Fanuc TP program (LS listing): layer_8.ls

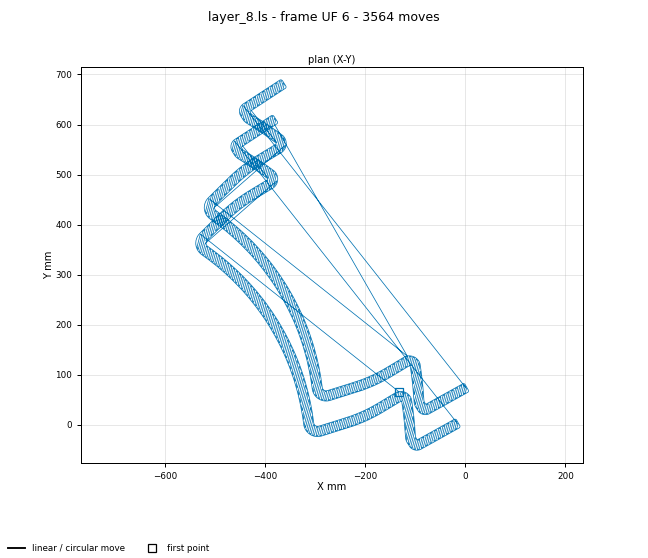
[picture p0: tool path of layer_8.ls in frame UF 6, 3564 of 3564 moves have a stored position in this frame; points joined in program order, loops and branches not executed]
/PROG layer_8
/ATTR
OWNER       = MNEDITOR;
CREATE      = DATE 100-11-20  TIME 09:43:21;
MODIFIED    = DATE 100-12-05  TIME 05:26:29;
LINE_COUNT = 1792;
PROTECT     = READ_WRITE;
TCD:  STACK_SIZE    = 0,
      TASK_PRIORITY = 50,
      TIME_SLICE    = 0,
      BUSY_LAMP_OFF = 0,
      ABORT_REQUEST = 0,
      PAUSE_REQUEST = 0;
DEFAULT_GROUP   = 1,1,*,*,*;
CONTROL_CODE    = 00000000 00000000;
/MN
:R[35]=79.0;
:R[34]=0;
1: L P[1] 240cm/min CNT100 COORD ;
: Arc Start[1];
2: L P[2] 240cm/min CNT100 COORD PTH ;
3: L P[3] 240cm/min CNT100 COORD PTH ;
4: L P[4] 240cm/min CNT100 COORD PTH ;
5: L P[5] 240cm/min CNT100 COORD PTH ;
6: L P[6] 240cm/min CNT100 COORD PTH ;
7: L P[7] 240cm/min CNT100 COORD PTH ;
8: L P[8] 240cm/min CNT100 COORD PTH ;
9: L P[9] 240cm/min CNT100 COORD PTH ;
10: L P[10] 240cm/min CNT100 COORD PTH ;
11: L P[11] 240cm/min CNT100 COORD PTH ;
12: L P[12] 240cm/min CNT100 COORD PTH ;
13: L P[13] 240cm/min CNT100 COORD PTH ;
14: L P[14] 240cm/min CNT100 COORD PTH ;
15: L P[15] 240cm/min CNT100 COORD PTH ;
16: L P[16] 240cm/min CNT100 COORD PTH ;
17: L P[17] 240cm/min CNT100 COORD PTH ;
18: L P[18] 240cm/min CNT100 COORD PTH ;
19: L P[19] 240cm/min CNT100 COORD PTH ;
20: L P[20] 240cm/min CNT100 COORD PTH ;
21: L P[21] 240cm/min CNT100 COORD PTH ;
22: L P[22] 240cm/min CNT100 COORD PTH ;
23: L P[23] 240cm/min CNT100 COORD PTH ;
24: L P[24] 240cm/min CNT100 COORD PTH ;
25: L P[25] 240cm/min CNT100 COORD PTH ;
26: L P[26] 240cm/min CNT100 COORD PTH ;
27: L P[27] 240cm/min CNT100 COORD PTH ;
28: L P[28] 240cm/min CNT100 COORD PTH ;
29: L P[29] 240cm/min CNT100 COORD PTH ;
30: L P[30] 240cm/min CNT100 COORD PTH ;
31: L P[31] 240cm/min CNT100 COORD PTH ;
32: L P[32] 240cm/min CNT100 COORD PTH ;
33: L P[33] 240cm/min CNT100 COORD PTH ;
34: L P[34] 240cm/min CNT100 COORD PTH ;
35: L P[35] 240cm/min CNT100 COORD PTH ;
36: L P[36] 240cm/min CNT100 COORD PTH ;
37: L P[37] 240cm/min CNT100 COORD PTH ;
38: L P[38] 240cm/min CNT100 COORD PTH ;
39: L P[39] 240cm/min CNT100 COORD PTH ;
40: L P[40] 240cm/min CNT100 COORD PTH ;
41: L P[41] 240cm/min CNT100 COORD PTH ;
42: L P[42] 240cm/min CNT100 COORD PTH ;
43: L P[43] 240cm/min CNT100 COORD PTH ;
44: L P[44] 240cm/min CNT100 COORD PTH ;
45: L P[45] 240cm/min CNT100 COORD PTH ;
46: L P[46] 240cm/min CNT100 COORD PTH ;
47: L P[47] 240cm/min CNT100 COORD PTH ;
48: L P[48] 240cm/min CNT100 COORD PTH ;
49: L P[49] 240cm/min CNT100 COORD PTH ;
50: L P[50] 240cm/min CNT100 COORD PTH ;
51: L P[51] 240cm/min CNT100 COORD PTH ;
52: L P[52] 240cm/min CNT100 COORD PTH ;
53: L P[53] 240cm/min CNT100 COORD PTH ;
54: L P[54] 240cm/min CNT100 COORD PTH ;
55: L P[55] 240cm/min CNT100 COORD PTH ;
56: L P[56] 240cm/min CNT100 COORD PTH ;
57: L P[57] 240cm/min CNT100 COORD PTH ;
58: L P[58] 240cm/min CNT100 COORD PTH ;
59: L P[59] 240cm/min CNT100 COORD PTH ;
60: L P[60] 240cm/min CNT100 COORD PTH ;
61: L P[61] 240cm/min CNT100 COORD PTH ;
62: L P[62] 240cm/min CNT100 COORD PTH ;
63: L P[63] 240cm/min CNT100 COORD PTH ;
64: L P[64] 240cm/min CNT100 COORD PTH ;
65: L P[65] 240cm/min CNT100 COORD PTH ;
66: L P[66] 240cm/min CNT100 COORD PTH ;
67: L P[67] 240cm/min CNT100 COORD PTH ;
68: L P[68] 240cm/min CNT100 COORD PTH ;
69: L P[69] 240cm/min CNT100 COORD PTH ;
70: L P[70] 240cm/min CNT100 COORD PTH ;
71: L P[71] 240cm/min CNT100 COORD PTH ;
72: L P[72] 240cm/min CNT100 COORD PTH ;
73: L P[73] 240cm/min CNT100 COORD PTH ;
74: L P[74] 240cm/min CNT100 COORD PTH ;
75: L P[75] 240cm/min CNT100 COORD PTH ;
76: L P[76] 240cm/min CNT100 COORD PTH ;
77: L P[77] 240cm/min CNT100 COORD PTH ;
78: L P[78] 240cm/min CNT100 COORD PTH ;
79: L P[79] 240cm/min CNT100 COORD PTH ;
80: L P[80] 240cm/min CNT100 COORD PTH ;
81: L P[81] 240cm/min CNT100 COORD PTH ;
82: L P[82] 240cm/min CNT100 COORD PTH ;
83: L P[83] 240cm/min CNT100 COORD PTH ;
84: L P[84] 240cm/min CNT100 COORD PTH ;
85: L P[85] 240cm/min CNT100 COORD PTH ;
86: L P[86] 240cm/min CNT100 COORD PTH ;
87: L P[87] 240cm/min CNT100 COORD PTH ;
88: L P[88] 240cm/min CNT100 COORD PTH ;
89: L P[89] 240cm/min CNT100 COORD PTH ;
90: L P[90] 240cm/min CNT100 COORD PTH ;
91: L P[91] 240cm/min CNT100 COORD PTH ;
92: L P[92] 240cm/min CNT100 COORD PTH ;
93: L P[93] 240cm/min CNT100 COORD PTH ;
94: L P[94] 240cm/min CNT100 COORD PTH ;
95: L P[95] 240cm/min CNT100 COORD PTH ;
96: L P[96] 240cm/min CNT100 COORD PTH ;
97: L P[97] 240cm/min CNT100 COORD PTH ;
98: L P[98] 240cm/min CNT100 COORD PTH ;
99: L P[99] 240cm/min CNT100 COORD PTH ;
100: L P[100] 240cm/min CNT100 COORD PTH ;
101: L P[101] 240cm/min CNT100 COORD PTH ;
102: L P[102] 240cm/min CNT100 COORD PTH ;
103: L P[103] 240cm/min CNT100 COORD PTH ;
104: L P[104] 240cm/min CNT100 COORD PTH ;
105: L P[105] 240cm/min CNT100 COORD PTH ;
106: L P[106] 240cm/min CNT100 COORD PTH ;
107: L P[107] 240cm/min CNT100 COORD PTH ;
108: L P[108] 240cm/min CNT100 COORD PTH ;
109: L P[109] 240cm/min CNT100 COORD PTH ;
110: L P[110] 240cm/min CNT100 COORD PTH ;
111: L P[111] 240cm/min CNT100 COORD PTH ;
112: L P[112] 240cm/min CNT100 COORD PTH ;
113: L P[113] 240cm/min CNT100 COORD PTH ;
114: L P[114] 240cm/min CNT100 COORD PTH ;
115: L P[115] 240cm/min CNT100 COORD PTH ;
116: L P[116] 240cm/min CNT100 COORD PTH ;
117: L P[117] 240cm/min CNT100 COORD PTH ;
118: L P[118] 240cm/min CNT100 COORD PTH ;
119: L P[119] 240cm/min CNT100 COORD PTH ;
120: L P[120] 240cm/min CNT100 COORD PTH ;
121: L P[121] 240cm/min CNT100 COORD PTH ;
122: L P[122] 240cm/min CNT100 COORD PTH ;
123: L P[123] 240cm/min CNT100 COORD PTH ;
124: L P[124] 240cm/min CNT100 COORD PTH ;
125: L P[125] 240cm/min CNT100 COORD PTH ;
126: L P[126] 240cm/min CNT100 COORD PTH ;
127: L P[127] 240cm/min CNT100 COORD PTH ;
128: L P[128] 240cm/min CNT100 COORD PTH ;
129: L P[129] 240cm/min CNT100 COORD PTH ;
130: L P[130] 240cm/min CNT100 COORD PTH ;
131: L P[131] 240cm/min CNT100 COORD PTH ;
132: L P[132] 240cm/min CNT100 COORD PTH ;
133: L P[133] 240cm/min CNT100 COORD PTH ;
134: L P[134] 240cm/min CNT100 COORD PTH ;
135: L P[135] 240cm/min CNT100 COORD PTH ;
136: L P[136] 240cm/min CNT100 COORD PTH ;
137: L P[137] 240cm/min CNT100 COORD PTH ;
138: L P[138] 240cm/min CNT100 COORD PTH ;
139: L P[139] 240cm/min CNT100 COORD PTH ;
140: L P[140] 240cm/min CNT100 COORD PTH ;
141: L P[141] 240cm/min CNT100 COORD PTH ;
142: L P[142] 240cm/min CNT100 COORD PTH ;
143: L P[143] 240cm/min CNT100 COORD PTH ;
144: L P[144] 240cm/min CNT100 COORD PTH ;
145: L P[145] 240cm/min CNT100 COORD PTH ;
146: L P[146] 240cm/min CNT100 COORD PTH ;
147: L P[147] 240cm/min CNT100 COORD PTH ;
148: L P[148] 240cm/min CNT100 COORD PTH ;
149: L P[149] 240cm/min CNT100 COORD PTH ;
150: L P[150] 240cm/min CNT100 COORD PTH ;
151: L P[151] 240cm/min CNT100 COORD PTH ;
152: L P[152] 240cm/min CNT100 COORD PTH ;
153: L P[153] 240cm/min CNT100 COORD PTH ;
154: L P[154] 240cm/min CNT100 COORD PTH ;
155: L P[155] 240cm/min CNT100 COORD PTH ;
156: L P[156] 240cm/min CNT100 COORD PTH ;
157: L P[157] 240cm/min CNT100 COORD PTH ;
158: L P[158] 240cm/min CNT100 COORD PTH ;
159: L P[159] 240cm/min CNT100 COORD PTH ;
160: L P[160] 240cm/min CNT100 COORD PTH ;
161: L P[161] 240cm/min CNT100 COORD PTH ;
162: L P[162] 240cm/min CNT100 COORD PTH ;
163: L P[163] 240cm/min CNT100 COORD PTH ;
164: L P[164] 240cm/min CNT100 COORD PTH ;
165: L P[165] 240cm/min CNT100 COORD PTH ;
166: L P[166] 240cm/min CNT100 COORD PTH ;
167: L P[167] 240cm/min CNT100 COORD PTH ;
168: L P[168] 240cm/min CNT100 COORD PTH ;
169: L P[169] 240cm/min CNT100 COORD PTH ;
170: L P[170] 240cm/min CNT100 COORD PTH ;
171: L P[171] 240cm/min CNT100 COORD PTH ;
172: L P[172] 240cm/min CNT100 COORD PTH ;
173: L P[173] 240cm/min CNT100 COORD PTH ;
174: L P[174] 240cm/min CNT100 COORD PTH ;
175: L P[175] 240cm/min CNT100 COORD PTH ;
176: L P[176] 240cm/min CNT100 COORD PTH ;
177: L P[177] 240cm/min CNT100 COORD PTH ;
178: L P[178] 240cm/min CNT100 COORD PTH ;
179: L P[179] 240cm/min CNT100 COORD PTH ;
180: L P[180] 240cm/min CNT100 COORD PTH ;
181: L P[181] 240cm/min CNT100 COORD PTH ;
182: L P[182] 240cm/min CNT100 COORD PTH ;
183: L P[183] 240cm/min CNT100 COORD PTH ;
184: L P[184] 240cm/min CNT100 COORD PTH ;
185: L P[185] 240cm/min CNT100 COORD PTH ;
186: L P[186] 240cm/min CNT100 COORD PTH ;
187: L P[187] 240cm/min CNT100 COORD PTH ;
188: L P[188] 240cm/min CNT100 COORD PTH ;
189: L P[189] 240cm/min CNT100 COORD PTH ;
190: L P[190] 240cm/min CNT100 COORD PTH ;
191: L P[191] 240cm/min CNT100 COORD PTH ;
192: L P[192] 240cm/min CNT100 COORD PTH ;
193: L P[193] 240cm/min CNT100 COORD PTH ;
194: L P[194] 240cm/min CNT100 COORD PTH ;
195: L P[195] 240cm/min CNT100 COORD PTH ;
196: L P[196] 240cm/min CNT100 COORD PTH ;
197: L P[197] 240cm/min CNT100 COORD PTH ;
198: L P[198] 240cm/min CNT100 COORD PTH ;
199: L P[199] 240cm/min CNT100 COORD PTH ;
200: L P[200] 240cm/min CNT100 COORD PTH ;
201: L P[201] 240cm/min CNT100 COORD PTH ;
202: L P[202] 240cm/min CNT100 COORD PTH ;
203: L P[203] 240cm/min CNT100 COORD PTH ;
204: L P[204] 240cm/min CNT100 COORD PTH ;
205: L P[205] 240cm/min CNT100 COORD PTH ;
206: L P[206] 240cm/min CNT100 COORD PTH ;
207: L P[207] 240cm/min CNT100 COORD PTH ;
208: L P[208] 240cm/min CNT100 COORD PTH ;
209: L P[209] 240cm/min CNT100 COORD PTH ;
210: L P[210] 240cm/min CNT100 COORD PTH ;
211: L P[211] 240cm/min CNT100 COORD PTH ;
212: L P[212] 240cm/min CNT100 COORD PTH ;
213: L P[213] 240cm/min CNT100 COORD PTH ;
214: L P[214] 240cm/min CNT100 COORD PTH ;
215: L P[215] 240cm/min CNT100 COORD PTH ;
216: L P[216] 240cm/min CNT100 COORD PTH ;
217: L P[217] 240cm/min CNT100 COORD PTH ;
218: L P[218] 240cm/min CNT100 COORD PTH ;
219: L P[219] 240cm/min CNT100 COORD PTH ;
220: L P[220] 240cm/min CNT100 COORD PTH ;
221: L P[221] 240cm/min CNT100 COORD PTH ;
222: L P[222] 240cm/min CNT100 COORD PTH ;
223: L P[223] 240cm/min CNT100 COORD PTH ;
224: L P[224] 240cm/min CNT100 COORD PTH ;
225: L P[225] 240cm/min CNT100 COORD PTH ;
226: L P[226] 240cm/min CNT100 COORD PTH ;
227: L P[227] 240cm/min CNT100 COORD PTH ;
228: L P[228] 240cm/min CNT100 COORD PTH ;
229: L P[229] 240cm/min CNT100 COORD PTH ;
230: L P[230] 240cm/min CNT100 COORD PTH ;
231: L P[231] 240cm/min CNT100 COORD PTH ;
232: L P[232] 240cm/min CNT100 COORD PTH ;
233: L P[233] 240cm/min CNT100 COORD PTH ;
234: L P[234] 240cm/min CNT100 COORD PTH ;
235: L P[235] 240cm/min CNT100 COORD PTH ;
236: L P[236] 240cm/min CNT100 COORD PTH ;
237: L P[237] 240cm/min CNT100 COORD PTH ;
238: L P[238] 240cm/min CNT100 COORD PTH ;
239: L P[239] 240cm/min CNT100 COORD PTH ;
240: L P[240] 240cm/min CNT100 COORD PTH ;
241: L P[241] 240cm/min CNT100 COORD PTH ;
242: L P[242] 240cm/min CNT100 COORD PTH ;
243: L P[243] 240cm/min CNT100 COORD PTH ;
244: L P[244] 240cm/min CNT100 COORD PTH ;
245: L P[245] 240cm/min CNT100 COORD PTH ;
246: L P[246] 240cm/min CNT100 COORD PTH ;
247: L P[247] 240cm/min CNT100 COORD PTH ;
248: L P[248] 240cm/min CNT100 COORD PTH ;
249: L P[249] 240cm/min CNT100 COORD PTH ;
250: L P[250] 240cm/min CNT100 COORD PTH ;
251: L P[251] 240cm/min CNT100 COORD PTH ;
252: L P[252] 240cm/min CNT100 COORD PTH ;
253: L P[253] 240cm/min CNT100 COORD PTH ;
254: L P[254] 240cm/min CNT100 COORD PTH ;
255: L P[255] 240cm/min CNT100 COORD PTH ;
256: L P[256] 240cm/min CNT100 COORD PTH ;
257: L P[257] 240cm/min CNT100 COORD PTH ;
258: L P[258] 240cm/min CNT100 COORD PTH ;
259: L P[259] 240cm/min CNT100 COORD PTH ;
260: L P[260] 240cm/min CNT100 COORD PTH ;
261: L P[261] 240cm/min CNT100 COORD PTH ;
262: L P[262] 240cm/min CNT100 COORD PTH ;
263: L P[263] 240cm/min CNT100 COORD PTH ;
264: L P[264] 240cm/min CNT100 COORD PTH ;
265: L P[265] 240cm/min CNT100 COORD PTH ;
266: L P[266] 240cm/min CNT100 COORD PTH ;
267: L P[267] 240cm/min CNT100 COORD PTH ;
268: L P[268] 240cm/min CNT100 COORD PTH ;
269: L P[269] 240cm/min CNT100 COORD PTH ;
270: L P[270] 240cm/min CNT100 COORD PTH ;
271: L P[271] 240cm/min CNT100 COORD PTH ;
272: L P[272] 240cm/min CNT100 COORD PTH ;
273: L P[273] 240cm/min CNT100 COORD PTH ;
274: L P[274] 240cm/min CNT100 COORD PTH ;
275: L P[275] 240cm/min CNT100 COORD PTH ;
276: L P[276] 240cm/min CNT100 COORD PTH ;
277: L P[277] 240cm/min CNT100 COORD PTH ;
278: L P[278] 240cm/min CNT100 COORD PTH ;
279: L P[279] 240cm/min CNT100 COORD PTH ;
280: L P[280] 240cm/min CNT100 COORD PTH ;
281: L P[281] 240cm/min CNT100 COORD PTH ;
282: L P[282] 240cm/min CNT100 COORD PTH ;
283: L P[283] 240cm/min CNT100 COORD PTH ;
284: L P[284] 240cm/min CNT100 COORD PTH ;
285: L P[285] 240cm/min CNT100 COORD PTH ;
286: L P[286] 240cm/min CNT100 COORD PTH ;
287: L P[287] 240cm/min CNT100 COORD PTH ;
288: L P[288] 240cm/min CNT100 COORD PTH ;
289: L P[289] 240cm/min CNT100 COORD PTH ;
290: L P[290] 240cm/min CNT100 COORD PTH ;
291: L P[291] 240cm/min CNT100 COORD PTH ;
292: L P[292] 240cm/min CNT100 COORD PTH ;
293: L P[293] 240cm/min CNT100 COORD PTH ;
294: L P[294] 240cm/min CNT100 COORD PTH ;
295: L P[295] 240cm/min CNT100 COORD PTH ;
296: L P[296] 240cm/min CNT100 COORD PTH ;
297: L P[297] 240cm/min CNT100 COORD PTH ;
298: L P[298] 240cm/min CNT100 COORD PTH ;
299: L P[299] 240cm/min CNT100 COORD PTH ;
300: L P[300] 240cm/min CNT100 COORD PTH ;
301: L P[301] 240cm/min CNT100 COORD PTH ;
302: L P[302] 240cm/min CNT100 COORD PTH ;
303: L P[303] 240cm/min CNT100 COORD PTH ;
304: L P[304] 240cm/min CNT100 COORD PTH ;
305: L P[305] 240cm/min CNT100 COORD PTH ;
306: L P[306] 240cm/min CNT100 COORD PTH ;
307: L P[307] 240cm/min CNT100 COORD PTH ;
308: L P[308] 240cm/min CNT100 COORD PTH ;
309: L P[309] 240cm/min CNT100 COORD PTH ;
310: L P[310] 240cm/min CNT100 COORD PTH ;
311: L P[311] 240cm/min CNT100 COORD PTH ;
312: L P[312] 240cm/min CNT100 COORD PTH ;
313: L P[313] 240cm/min CNT100 COORD PTH ;
314: L P[314] 240cm/min CNT100 COORD PTH ;
315: L P[315] 240cm/min CNT100 COORD PTH ;
316: L P[316] 240cm/min CNT100 COORD PTH ;
317: L P[317] 240cm/min CNT100 COORD PTH ;
318: L P[318] 240cm/min CNT100 COORD PTH ;
319: L P[319] 240cm/min CNT100 COORD PTH ;
320: L P[320] 240cm/min CNT100 COORD PTH ;
321: L P[321] 240cm/min CNT100 COORD PTH ;
322: L P[322] 240cm/min CNT100 COORD PTH ;
323: L P[323] 240cm/min CNT100 COORD PTH ;
324: L P[324] 240cm/min CNT100 COORD PTH ;
325: L P[325] 240cm/min CNT100 COORD PTH ;
326: L P[326] 240cm/min CNT100 COORD PTH ;
327: L P[327] 240cm/min CNT100 COORD PTH ;
328: L P[328] 240cm/min CNT100 COORD PTH ;
329: L P[329] 240cm/min CNT100 COORD PTH ;
330: L P[330] 240cm/min CNT100 COORD PTH ;
331: L P[331] 240cm/min CNT100 COORD PTH ;
332: L P[332] 240cm/min CNT100 COORD PTH ;
333: L P[333] 240cm/min CNT100 COORD PTH ;
334: L P[334] 240cm/min CNT100 COORD PTH ;
335: L P[335] 240cm/min CNT100 COORD PTH ;
336: L P[336] 240cm/min CNT100 COORD PTH ;
337: L P[337] 240cm/min CNT100 COORD PTH ;
338: L P[338] 240cm/min CNT100 COORD PTH ;
339: L P[339] 240cm/min CNT100 COORD PTH ;
340: L P[340] 240cm/min CNT100 COORD PTH ;
341: L P[341] 240cm/min CNT100 COORD PTH ;
342: L P[342] 240cm/min CNT100 COORD PTH ;
343: L P[343] 240cm/min CNT100 COORD PTH ;
344: L P[344] 240cm/min CNT100 COORD PTH ;
345: L P[345] 240cm/min CNT100 COORD PTH ;
346: L P[346] 240cm/min CNT100 COORD PTH ;
347: L P[347] 240cm/min CNT100 COORD PTH ;
348: L P[348] 240cm/min CNT100 COORD PTH ;
349: L P[349] 240cm/min CNT100 COORD PTH ;
350: L P[350] 240cm/min CNT100 COORD PTH ;
351: L P[351] 240cm/min CNT100 COORD PTH ;
352: L P[352] 240cm/min CNT100 COORD PTH ;
353: L P[353] 240cm/min CNT100 COORD PTH ;
354: L P[354] 240cm/min CNT100 COORD PTH ;
355: L P[355] 240cm/min CNT100 COORD PTH ;
356: L P[356] 240cm/min CNT100 COORD PTH ;
357: L P[357] 240cm/min CNT100 COORD PTH ;
358: L P[358] 240cm/min CNT100 COORD PTH ;
359: L P[359] 240cm/min CNT100 COORD PTH ;
360: L P[360] 240cm/min CNT100 COORD PTH ;
361: L P[361] 240cm/min CNT100 COORD PTH ;
362: L P[362] 240cm/min CNT100 COORD PTH ;
363: L P[363] 240cm/min CNT100 COORD PTH ;
364: L P[364] 240cm/min CNT100 COORD PTH ;
365: L P[365] 240cm/min CNT100 COORD PTH ;
366: L P[366] 240cm/min CNT100 COORD PTH ;
367: L P[367] 240cm/min CNT100 COORD PTH ;
368: L P[368] 240cm/min CNT100 COORD PTH ;
369: L P[369] 240cm/min CNT100 COORD PTH ;
370: L P[370] 240cm/min CNT100 COORD PTH ;
371: L P[371] 240cm/min CNT100 COORD PTH ;
372: L P[372] 240cm/min CNT100 COORD PTH ;
373: L P[373] 240cm/min CNT100 COORD PTH ;
374: L P[374] 240cm/min CNT100 COORD PTH ;
375: L P[375] 240cm/min CNT100 COORD PTH ;
376: L P[376] 240cm/min CNT100 COORD PTH ;
377: L P[377] 240cm/min CNT100 COORD PTH ;
378: L P[378] 240cm/min CNT100 COORD PTH ;
379: L P[379] 240cm/min CNT100 COORD PTH ;
380: L P[380] 240cm/min CNT100 COORD PTH ;
381: L P[381] 240cm/min CNT100 COORD PTH ;
382: L P[382] 240cm/min CNT100 COORD PTH ;
383: L P[383] 240cm/min CNT100 COORD PTH ;
384: L P[384] 240cm/min CNT100 COORD PTH ;
385: L P[385] 240cm/min CNT100 COORD PTH ;
386: L P[386] 240cm/min CNT100 COORD PTH ;
387: L P[387] 240cm/min CNT100 COORD PTH ;
388: L P[388] 240cm/min CNT100 COORD PTH ;
389: L P[389] 240cm/min CNT100 COORD PTH ;
390: L P[390] 240cm/min CNT100 COORD PTH ;
391: L P[391] 240cm/min CNT100 COORD PTH ;
392: L P[392] 240cm/min CNT100 COORD PTH ;
393: L P[393] 240cm/min CNT100 COORD PTH ;
394: L P[394] 240cm/min CNT100 COORD PTH ;
395: L P[395] 240cm/min CNT100 COORD PTH ;
396: L P[396] 240cm/min CNT100 COORD PTH ;
397: L P[397] 240cm/min CNT100 COORD PTH ;
398: L P[398] 240cm/min CNT100 COORD PTH ;
399: L P[399] 240cm/min CNT100 COORD PTH ;
: Arc End[1];
400: L P[400] 240cm/min CNT100 COORD ;
: Arc Start[1];
401: L P[401] 240cm/min CNT100 COORD PTH ;
402: L P[402] 240cm/min CNT100 COORD PTH ;
403: L P[403] 240cm/min CNT100 COORD PTH ;
404: L P[404] 240cm/min CNT100 COORD PTH ;
405: L P[405] 240cm/min CNT100 COORD PTH ;
406: L P[406] 240cm/min CNT100 COORD PTH ;
407: L P[407] 240cm/min CNT100 COORD PTH ;
408: L P[408] 240cm/min CNT100 COORD PTH ;
409: L P[409] 240cm/min CNT100 COORD PTH ;
410: L P[410] 240cm/min CNT100 COORD PTH ;
411: L P[411] 240cm/min CNT100 COORD PTH ;
412: L P[412] 240cm/min CNT100 COORD PTH ;
413: L P[413] 240cm/min CNT100 COORD PTH ;
414: L P[414] 240cm/min CNT100 COORD PTH ;
415: L P[415] 240cm/min CNT100 COORD PTH ;
416: L P[416] 240cm/min CNT100 COORD PTH ;
417: L P[417] 240cm/min CNT100 COORD PTH ;
418: L P[418] 240cm/min CNT100 COORD PTH ;
419: L P[419] 240cm/min CNT100 COORD PTH ;
420: L P[420] 240cm/min CNT100 COORD PTH ;
421: L P[421] 240cm/min CNT100 COORD PTH ;
422: L P[422] 240cm/min CNT100 COORD PTH ;
423: L P[423] 240cm/min CNT100 COORD PTH ;
424: L P[424] 240cm/min CNT100 COORD PTH ;
425: L P[425] 240cm/min CNT100 COORD PTH ;
426: L P[426] 240cm/min CNT100 COORD PTH ;
427: L P[427] 240cm/min CNT100 COORD PTH ;
428: L P[428] 240cm/min CNT100 COORD PTH ;
429: L P[429] 240cm/min CNT100 COORD PTH ;
430: L P[430] 240cm/min CNT100 COORD PTH ;
431: L P[431] 240cm/min CNT100 COORD PTH ;
432: L P[432] 240cm/min CNT100 COORD PTH ;
433: L P[433] 240cm/min CNT100 COORD PTH ;
434: L P[434] 240cm/min CNT100 COORD PTH ;
435: L P[435] 240cm/min CNT100 COORD PTH ;
436: L P[436] 240cm/min CNT100 COORD PTH ;
437: L P[437] 240cm/min CNT100 COORD PTH ;
438: L P[438] 240cm/min CNT100 COORD PTH ;
439: L P[439] 240cm/min CNT100 COORD PTH ;
440: L P[440] 240cm/min CNT100 COORD PTH ;
441: L P[441] 240cm/min CNT100 COORD PTH ;
442: L P[442] 240cm/min CNT100 COORD PTH ;
443: L P[443] 240cm/min CNT100 COORD PTH ;
444: L P[444] 240cm/min CNT100 COORD PTH ;
445: L P[445] 240cm/min CNT100 COORD PTH ;
446: L P[446] 240cm/min CNT100 COORD PTH ;
447: L P[447] 240cm/min CNT100 COORD PTH ;
448: L P[448] 240cm/min CNT100 COORD PTH ;
449: L P[449] 240cm/min CNT100 COORD PTH ;
450: L P[450] 240cm/min CNT100 COORD PTH ;
451: L P[451] 240cm/min CNT100 COORD PTH ;
452: L P[452] 240cm/min CNT100 COORD PTH ;
453: L P[453] 240cm/min CNT100 COORD PTH ;
454: L P[454] 240cm/min CNT100 COORD PTH ;
455: L P[455] 240cm/min CNT100 COORD PTH ;
456: L P[456] 240cm/min CNT100 COORD PTH ;
457: L P[457] 240cm/min CNT100 COORD PTH ;
458: L P[458] 240cm/min CNT100 COORD PTH ;
459: L P[459] 240cm/min CNT100 COORD PTH ;
460: L P[460] 240cm/min CNT100 COORD PTH ;
461: L P[461] 240cm/min CNT100 COORD PTH ;
462: L P[462] 240cm/min CNT100 COORD PTH ;
463: L P[463] 240cm/min CNT100 COORD PTH ;
464: L P[464] 240cm/min CNT100 COORD PTH ;
465: L P[465] 240cm/min CNT100 COORD PTH ;
466: L P[466] 240cm/min CNT100 COORD PTH ;
467: L P[467] 240cm/min CNT100 COORD PTH ;
468: L P[468] 240cm/min CNT100 COORD PTH ;
469: L P[469] 240cm/min CNT100 COORD PTH ;
470: L P[470] 240cm/min CNT100 COORD PTH ;
471: L P[471] 240cm/min CNT100 COORD PTH ;
472: L P[472] 240cm/min CNT100 COORD PTH ;
473: L P[473] 240cm/min CNT100 COORD PTH ;
474: L P[474] 240cm/min CNT100 COORD PTH ;
475: L P[475] 240cm/min CNT100 COORD PTH ;
476: L P[476] 240cm/min CNT100 COORD PTH ;
477: L P[477] 240cm/min CNT100 COORD PTH ;
478: L P[478] 240cm/min CNT100 COORD PTH ;
479: L P[479] 240cm/min CNT100 COORD PTH ;
480: L P[480] 240cm/min CNT100 COORD PTH ;
481: L P[481] 240cm/min CNT100 COORD PTH ;
482: L P[482] 240cm/min CNT100 COORD PTH ;
483: L P[483] 240cm/min CNT100 COORD PTH ;
484: L P[484] 240cm/min CNT100 COORD PTH ;
485: L P[485] 240cm/min CNT100 COORD PTH ;
486: L P[486] 240cm/min CNT100 COORD PTH ;
487: L P[487] 240cm/min CNT100 COORD PTH ;
488: L P[488] 240cm/min CNT100 COORD PTH ;
489: L P[489] 240cm/min CNT100 COORD PTH ;
490: L P[490] 240cm/min CNT100 COORD PTH ;
491: L P[491] 240cm/min CNT100 COORD PTH ;
492: L P[492] 240cm/min CNT100 COORD PTH ;
493: L P[493] 240cm/min CNT100 COORD PTH ;
494: L P[494] 240cm/min CNT100 COORD PTH ;
495: L P[495] 240cm/min CNT100 COORD PTH ;
496: L P[496] 240cm/min CNT100 COORD PTH ;
497: L P[497] 240cm/min CNT100 COORD PTH ;
498: L P[498] 240cm/min CNT100 COORD PTH ;
499: L P[499] 240cm/min CNT100 COORD PTH ;
500: L P[500] 240cm/min CNT100 COORD PTH ;
501: L P[501] 240cm/min CNT100 COORD PTH ;
502: L P[502] 240cm/min CNT100 COORD PTH ;
503: L P[503] 240cm/min CNT100 COORD PTH ;
504: L P[504] 240cm/min CNT100 COORD PTH ;
505: L P[505] 240cm/min CNT100 COORD PTH ;
506: L P[506] 240cm/min CNT100 COORD PTH ;
507: L P[507] 240cm/min CNT100 COORD PTH ;
508: L P[508] 240cm/min CNT100 COORD PTH ;
509: L P[509] 240cm/min CNT100 COORD PTH ;
510: L P[510] 240cm/min CNT100 COORD PTH ;
511: L P[511] 240cm/min CNT100 COORD PTH ;
512: L P[512] 240cm/min CNT100 COORD PTH ;
513: L P[513] 240cm/min CNT100 COORD PTH ;
514: L P[514] 240cm/min CNT100 COORD PTH ;
515: L P[515] 240cm/min CNT100 COORD PTH ;
516: L P[516] 240cm/min CNT100 COORD PTH ;
517: L P[517] 240cm/min CNT100 COORD PTH ;
518: L P[518] 240cm/min CNT100 COORD PTH ;
519: L P[519] 240cm/min CNT100 COORD PTH ;
520: L P[520] 240cm/min CNT100 COORD PTH ;
521: L P[521] 240cm/min CNT100 COORD PTH ;
522: L P[522] 240cm/min CNT100 COORD PTH ;
523: L P[523] 240cm/min CNT100 COORD PTH ;
524: L P[524] 240cm/min CNT100 COORD PTH ;
525: L P[525] 240cm/min CNT100 COORD PTH ;
526: L P[526] 240cm/min CNT100 COORD PTH ;
527: L P[527] 240cm/min CNT100 COORD PTH ;
528: L P[528] 240cm/min CNT100 COORD PTH ;
529: L P[529] 240cm/min CNT100 COORD PTH ;
530: L P[530] 240cm/min CNT100 COORD PTH ;
531: L P[531] 240cm/min CNT100 COORD PTH ;
532: L P[532] 240cm/min CNT100 COORD PTH ;
533: L P[533] 240cm/min CNT100 COORD PTH ;
534: L P[534] 240cm/min CNT100 COORD PTH ;
535: L P[535] 240cm/min CNT100 COORD PTH ;
536: L P[536] 240cm/min CNT100 COORD PTH ;
537: L P[537] 240cm/min CNT100 COORD PTH ;
538: L P[538] 240cm/min CNT100 COORD PTH ;
539: L P[539] 240cm/min CNT100 COORD PTH ;
540: L P[540] 240cm/min CNT100 COORD PTH ;
541: L P[541] 240cm/min CNT100 COORD PTH ;
542: L P[542] 240cm/min CNT100 COORD PTH ;
543: L P[543] 240cm/min CNT100 COORD PTH ;
544: L P[544] 240cm/min CNT100 COORD PTH ;
545: L P[545] 240cm/min CNT100 COORD PTH ;
546: L P[546] 240cm/min CNT100 COORD PTH ;
547: L P[547] 240cm/min CNT100 COORD PTH ;
548: L P[548] 240cm/min CNT100 COORD PTH ;
549: L P[549] 240cm/min CNT100 COORD PTH ;
550: L P[550] 240cm/min CNT100 COORD PTH ;
551: L P[551] 240cm/min CNT100 COORD PTH ;
552: L P[552] 240cm/min CNT100 COORD PTH ;
553: L P[553] 240cm/min CNT100 COORD PTH ;
554: L P[554] 240cm/min CNT100 COORD PTH ;
555: L P[555] 240cm/min CNT100 COORD PTH ;
556: L P[556] 240cm/min CNT100 COORD PTH ;
557: L P[557] 240cm/min CNT100 COORD PTH ;
558: L P[558] 240cm/min CNT100 COORD PTH ;
559: L P[559] 240cm/min CNT100 COORD PTH ;
560: L P[560] 240cm/min CNT100 COORD PTH ;
561: L P[561] 240cm/min CNT100 COORD PTH ;
562: L P[562] 240cm/min CNT100 COORD PTH ;
563: L P[563] 240cm/min CNT100 COORD PTH ;
564: L P[564] 240cm/min CNT100 COORD PTH ;
565: L P[565] 240cm/min CNT100 COORD PTH ;
566: L P[566] 240cm/min CNT100 COORD PTH ;
567: L P[567] 240cm/min CNT100 COORD PTH ;
568: L P[568] 240cm/min CNT100 COORD PTH ;
569: L P[569] 240cm/min CNT100 COORD PTH ;
570: L P[570] 240cm/min CNT100 COORD PTH ;
571: L P[571] 240cm/min CNT100 COORD PTH ;
572: L P[572] 240cm/min CNT100 COORD PTH ;
573: L P[573] 240cm/min CNT100 COORD PTH ;
574: L P[574] 240cm/min CNT100 COORD PTH ;
575: L P[575] 240cm/min CNT100 COORD PTH ;
576: L P[576] 240cm/min CNT100 COORD PTH ;
577: L P[577] 240cm/min CNT100 COORD PTH ;
578: L P[578] 240cm/min CNT100 COORD PTH ;
579: L P[579] 240cm/min CNT100 COORD PTH ;
580: L P[580] 240cm/min CNT100 COORD PTH ;
581: L P[581] 240cm/min CNT100 COORD PTH ;
582: L P[582] 240cm/min CNT100 COORD PTH ;
583: L P[583] 240cm/min CNT100 COORD PTH ;
584: L P[584] 240cm/min CNT100 COORD PTH ;
585: L P[585] 240cm/min CNT100 COORD PTH ;
586: L P[586] 240cm/min CNT100 COORD PTH ;
587: L P[587] 240cm/min CNT100 COORD PTH ;
588: L P[588] 240cm/min CNT100 COORD PTH ;
589: L P[589] 240cm/min CNT100 COORD PTH ;
590: L P[590] 240cm/min CNT100 COORD PTH ;
591: L P[591] 240cm/min CNT100 COORD PTH ;
592: L P[592] 240cm/min CNT100 COORD PTH ;
593: L P[593] 240cm/min CNT100 COORD PTH ;
594: L P[594] 240cm/min CNT100 COORD PTH ;
595: L P[595] 240cm/min CNT100 COORD PTH ;
596: L P[596] 240cm/min CNT100 COORD PTH ;
597: L P[597] 240cm/min CNT100 COORD PTH ;
598: L P[598] 240cm/min CNT100 COORD PTH ;
599: L P[599] 240cm/min CNT100 COORD PTH ;
600: L P[600] 240cm/min CNT100 COORD PTH ;
601: L P[601] 240cm/min CNT100 COORD PTH ;
602: L P[602] 240cm/min CNT100 COORD PTH ;
603: L P[603] 240cm/min CNT100 COORD PTH ;
604: L P[604] 240cm/min CNT100 COORD PTH ;
605: L P[605] 240cm/min CNT100 COORD PTH ;
606: L P[606] 240cm/min CNT100 COORD PTH ;
607: L P[607] 240cm/min CNT100 COORD PTH ;
608: L P[608] 240cm/min CNT100 COORD PTH ;
609: L P[609] 240cm/min CNT100 COORD PTH ;
610: L P[610] 240cm/min CNT100 COORD PTH ;
611: L P[611] 240cm/min CNT100 COORD PTH ;
612: L P[612] 240cm/min CNT100 COORD PTH ;
613: L P[613] 240cm/min CNT100 COORD PTH ;
614: L P[614] 240cm/min CNT100 COORD PTH ;
615: L P[615] 240cm/min CNT100 COORD PTH ;
616: L P[616] 240cm/min CNT100 COORD PTH ;
617: L P[617] 240cm/min CNT100 COORD PTH ;
618: L P[618] 240cm/min CNT100 COORD PTH ;
619: L P[619] 240cm/min CNT100 COORD PTH ;
620: L P[620] 240cm/min CNT100 COORD PTH ;
621: L P[621] 240cm/min CNT100 COORD PTH ;
622: L P[622] 240cm/min CNT100 COORD PTH ;
623: L P[623] 240cm/min CNT100 COORD PTH ;
624: L P[624] 240cm/min CNT100 COORD PTH ;
625: L P[625] 240cm/min CNT100 COORD PTH ;
626: L P[626] 240cm/min CNT100 COORD PTH ;
627: L P[627] 240cm/min CNT100 COORD PTH ;
628: L P[628] 240cm/min CNT100 COORD PTH ;
629: L P[629] 240cm/min CNT100 COORD PTH ;
630: L P[630] 240cm/min CNT100 COORD PTH ;
631: L P[631] 240cm/min CNT100 COORD PTH ;
632: L P[632] 240cm/min CNT100 COORD PTH ;
633: L P[633] 240cm/min CNT100 COORD PTH ;
634: L P[634] 240cm/min CNT100 COORD PTH ;
635: L P[635] 240cm/min CNT100 COORD PTH ;
636: L P[636] 240cm/min CNT100 COORD PTH ;
637: L P[637] 240cm/min CNT100 COORD PTH ;
638: L P[638] 240cm/min CNT100 COORD PTH ;
639: L P[639] 240cm/min CNT100 COORD PTH ;
640: L P[640] 240cm/min CNT100 COORD PTH ;
641: L P[641] 240cm/min CNT100 COORD PTH ;
642: L P[642] 240cm/min CNT100 COORD PTH ;
643: L P[643] 240cm/min CNT100 COORD PTH ;
644: L P[644] 240cm/min CNT100 COORD PTH ;
645: L P[645] 240cm/min CNT100 COORD PTH ;
646: L P[646] 240cm/min CNT100 COORD PTH ;
647: L P[647] 240cm/min CNT100 COORD PTH ;
648: L P[648] 240cm/min CNT100 COORD PTH ;
649: L P[649] 240cm/min CNT100 COORD PTH ;
650: L P[650] 240cm/min CNT100 COORD PTH ;
651: L P[651] 240cm/min CNT100 COORD PTH ;
652: L P[652] 240cm/min CNT100 COORD PTH ;
653: L P[653] 240cm/min CNT100 COORD PTH ;
654: L P[654] 240cm/min CNT100 COORD PTH ;
655: L P[655] 240cm/min CNT100 COORD PTH ;
656: L P[656] 240cm/min CNT100 COORD PTH ;
: Arc End[1];
657: L P[657] 240cm/min CNT100 COORD ;
: Arc Start[1];
658: L P[658] 240cm/min CNT100 COORD PTH ;
659: L P[659] 240cm/min CNT100 COORD PTH ;
660: L P[660] 240cm/min CNT100 COORD PTH ;
661: L P[661] 240cm/min CNT100 COORD PTH ;
662: L P[662] 240cm/min CNT100 COORD PTH ;
663: L P[663] 240cm/min CNT100 COORD PTH ;
664: L P[664] 240cm/min CNT100 COORD PTH ;
665: L P[665] 240cm/min CNT100 COORD PTH ;
666: L P[666] 240cm/min CNT100 COORD PTH ;
667: L P[667] 240cm/min CNT100 COORD PTH ;
668: L P[668] 240cm/min CNT100 COORD PTH ;
669: L P[669] 240cm/min CNT100 COORD PTH ;
670: L P[670] 240cm/min CNT100 COORD PTH ;
671: L P[671] 240cm/min CNT100 COORD PTH ;
672: L P[672] 240cm/min CNT100 COORD PTH ;
673: L P[673] 240cm/min CNT100 COORD PTH ;
674: L P[674] 240cm/min CNT100 COORD PTH ;
675: L P[675] 240cm/min CNT100 COORD PTH ;
676: L P[676] 240cm/min CNT100 COORD PTH ;
677: L P[677] 240cm/min CNT100 COORD PTH ;
678: L P[678] 240cm/min CNT100 COORD PTH ;
679: L P[679] 240cm/min CNT100 COORD PTH ;
680: L P[680] 240cm/min CNT100 COORD PTH ;
681: L P[681] 240cm/min CNT100 COORD PTH ;
682: L P[682] 240cm/min CNT100 COORD PTH ;
683: L P[683] 240cm/min CNT100 COORD PTH ;
684: L P[684] 240cm/min CNT100 COORD PTH ;
685: L P[685] 240cm/min CNT100 COORD PTH ;
686: L P[686] 240cm/min CNT100 COORD PTH ;
687: L P[687] 240cm/min CNT100 COORD PTH ;
688: L P[688] 240cm/min CNT100 COORD PTH ;
689: L P[689] 240cm/min CNT100 COORD PTH ;
690: L P[690] 240cm/min CNT100 COORD PTH ;
691: L P[691] 240cm/min CNT100 COORD PTH ;
692: L P[692] 240cm/min CNT100 COORD PTH ;
693: L P[693] 240cm/min CNT100 COORD PTH ;
694: L P[694] 240cm/min CNT100 COORD PTH ;
695: L P[695] 240cm/min CNT100 COORD PTH ;
696: L P[696] 240cm/min CNT100 COORD PTH ;
697: L P[697] 240cm/min CNT100 COORD PTH ;
698: L P[698] 240cm/min CNT100 COORD PTH ;
699: L P[699] 240cm/min CNT100 COORD PTH ;
700: L P[700] 240cm/min CNT100 COORD PTH ;
701: L P[701] 240cm/min CNT100 COORD PTH ;
702: L P[702] 240cm/min CNT100 COORD PTH ;
703: L P[703] 240cm/min CNT100 COORD PTH ;
704: L P[704] 240cm/min CNT100 COORD PTH ;
705: L P[705] 240cm/min CNT100 COORD PTH ;
706: L P[706] 240cm/min CNT100 COORD PTH ;
707: L P[707] 240cm/min CNT100 COORD PTH ;
708: L P[708] 240cm/min CNT100 COORD PTH ;
709: L P[709] 240cm/min CNT100 COORD PTH ;
710: L P[710] 240cm/min CNT100 COORD PTH ;
711: L P[711] 240cm/min CNT100 COORD PTH ;
712: L P[712] 240cm/min CNT100 COORD PTH ;
713: L P[713] 240cm/min CNT100 COORD PTH ;
714: L P[714] 240cm/min CNT100 COORD PTH ;
715: L P[715] 240cm/min CNT100 COORD PTH ;
716: L P[716] 240cm/min CNT100 COORD PTH ;
717: L P[717] 240cm/min CNT100 COORD PTH ;
718: L P[718] 240cm/min CNT100 COORD PTH ;
719: L P[719] 240cm/min CNT100 COORD PTH ;
720: L P[720] 240cm/min CNT100 COORD PTH ;
721: L P[721] 240cm/min CNT100 COORD PTH ;
722: L P[722] 240cm/min CNT100 COORD PTH ;
723: L P[723] 240cm/min CNT100 COORD PTH ;
724: L P[724] 240cm/min CNT100 COORD PTH ;
725: L P[725] 240cm/min CNT100 COORD PTH ;
726: L P[726] 240cm/min CNT100 COORD PTH ;
727: L P[727] 240cm/min CNT100 COORD PTH ;
728: L P[728] 240cm/min CNT100 COORD PTH ;
729: L P[729] 240cm/min CNT100 COORD PTH ;
730: L P[730] 240cm/min CNT100 COORD PTH ;
731: L P[731] 240cm/min CNT100 COORD PTH ;
732: L P[732] 240cm/min CNT100 COORD PTH ;
733: L P[733] 240cm/min CNT100 COORD PTH ;
734: L P[734] 240cm/min CNT100 COORD PTH ;
735: L P[735] 240cm/min CNT100 COORD PTH ;
736: L P[736] 240cm/min CNT100 COORD PTH ;
737: L P[737] 240cm/min CNT100 COORD PTH ;
738: L P[738] 240cm/min CNT100 COORD PTH ;
739: L P[739] 240cm/min CNT100 COORD PTH ;
740: L P[740] 240cm/min CNT100 COORD PTH ;
741: L P[741] 240cm/min CNT100 COORD PTH ;
742: L P[742] 240cm/min CNT100 COORD PTH ;
743: L P[743] 240cm/min CNT100 COORD PTH ;
744: L P[744] 240cm/min CNT100 COORD PTH ;
745: L P[745] 240cm/min CNT100 COORD PTH ;
746: L P[746] 240cm/min CNT100 COORD PTH ;
747: L P[747] 240cm/min CNT100 COORD PTH ;
748: L P[748] 240cm/min CNT100 COORD PTH ;
749: L P[749] 240cm/min CNT100 COORD PTH ;
750: L P[750] 240cm/min CNT100 COORD PTH ;
751: L P[751] 240cm/min CNT100 COORD PTH ;
752: L P[752] 240cm/min CNT100 COORD PTH ;
753: L P[753] 240cm/min CNT100 COORD PTH ;
754: L P[754] 240cm/min CNT100 COORD PTH ;
755: L P[755] 240cm/min CNT100 COORD PTH ;
756: L P[756] 240cm/min CNT100 COORD PTH ;
757: L P[757] 240cm/min CNT100 COORD PTH ;
758: L P[758] 240cm/min CNT100 COORD PTH ;
759: L P[759] 240cm/min CNT100 COORD PTH ;
760: L P[760] 240cm/min CNT100 COORD PTH ;
761: L P[761] 240cm/min CNT100 COORD PTH ;
762: L P[762] 240cm/min CNT100 COORD PTH ;
763: L P[763] 240cm/min CNT100 COORD PTH ;
764: L P[764] 240cm/min CNT100 COORD PTH ;
765: L P[765] 240cm/min CNT100 COORD PTH ;
766: L P[766] 240cm/min CNT100 COORD PTH ;
767: L P[767] 240cm/min CNT100 COORD PTH ;
768: L P[768] 240cm/min CNT100 COORD PTH ;
769: L P[769] 240cm/min CNT100 COORD PTH ;
770: L P[770] 240cm/min CNT100 COORD PTH ;
771: L P[771] 240cm/min CNT100 COORD PTH ;
772: L P[772] 240cm/min CNT100 COORD PTH ;
773: L P[773] 240cm/min CNT100 COORD PTH ;
774: L P[774] 240cm/min CNT100 COORD PTH ;
775: L P[775] 240cm/min CNT100 COORD PTH ;
776: L P[776] 240cm/min CNT100 COORD PTH ;
777: L P[777] 240cm/min CNT100 COORD PTH ;
778: L P[778] 240cm/min CNT100 COORD PTH ;
779: L P[779] 240cm/min CNT100 COORD PTH ;
780: L P[780] 240cm/min CNT100 COORD PTH ;
781: L P[781] 240cm/min CNT100 COORD PTH ;
782: L P[782] 240cm/min CNT100 COORD PTH ;
783: L P[783] 240cm/min CNT100 COORD PTH ;
784: L P[784] 240cm/min CNT100 COORD PTH ;
785: L P[785] 240cm/min CNT100 COORD PTH ;
786: L P[786] 240cm/min CNT100 COORD PTH ;
787: L P[787] 240cm/min CNT100 COORD PTH ;
788: L P[788] 240cm/min CNT100 COORD PTH ;
789: L P[789] 240cm/min CNT100 COORD PTH ;
790: L P[790] 240cm/min CNT100 COORD PTH ;
791: L P[791] 240cm/min CNT100 COORD PTH ;
792: L P[792] 240cm/min CNT100 COORD PTH ;
793: L P[793] 240cm/min CNT100 COORD PTH ;
794: L P[794] 240cm/min CNT100 COORD PTH ;
795: L P[795] 240cm/min CNT100 COORD PTH ;
796: L P[796] 240cm/min CNT100 COORD PTH ;
797: L P[797] 240cm/min CNT100 COORD PTH ;
798: L P[798] 240cm/min CNT100 COORD PTH ;
799: L P[799] 240cm/min CNT100 COORD PTH ;
800: L P[800] 240cm/min CNT100 COORD PTH ;
801: L P[801] 240cm/min CNT100 COORD PTH ;
802: L P[802] 240cm/min CNT100 COORD PTH ;
803: L P[803] 240cm/min CNT100 COORD PTH ;
804: L P[804] 240cm/min CNT100 COORD PTH ;
805: L P[805] 240cm/min CNT100 COORD PTH ;
806: L P[806] 240cm/min CNT100 COORD PTH ;
807: L P[807] 240cm/min CNT100 COORD PTH ;
808: L P[808] 240cm/min CNT100 COORD PTH ;
809: L P[809] 240cm/min CNT100 COORD PTH ;
810: L P[810] 240cm/min CNT100 COORD PTH ;
811: L P[811] 240cm/min CNT100 COORD PTH ;
812: L P[812] 240cm/min CNT100 COORD PTH ;
813: L P[813] 240cm/min CNT100 COORD PTH ;
814: L P[814] 240cm/min CNT100 COORD PTH ;
815: L P[815] 240cm/min CNT100 COORD PTH ;
816: L P[816] 240cm/min CNT100 COORD PTH ;
817: L P[817] 240cm/min CNT100 COORD PTH ;
818: L P[818] 240cm/min CNT100 COORD PTH ;
819: L P[819] 240cm/min CNT100 COORD PTH ;
820: L P[820] 240cm/min CNT100 COORD PTH ;
821: L P[821] 240cm/min CNT100 COORD PTH ;
822: L P[822] 240cm/min CNT100 COORD PTH ;
823: L P[823] 240cm/min CNT100 COORD PTH ;
824: L P[824] 240cm/min CNT100 COORD PTH ;
825: L P[825] 240cm/min CNT100 COORD PTH ;
826: L P[826] 240cm/min CNT100 COORD PTH ;
827: L P[827] 240cm/min CNT100 COORD PTH ;
828: L P[828] 240cm/min CNT100 COORD PTH ;
829: L P[829] 240cm/min CNT100 COORD PTH ;
830: L P[830] 240cm/min CNT100 COORD PTH ;
831: L P[831] 240cm/min CNT100 COORD PTH ;
832: L P[832] 240cm/min CNT100 COORD PTH ;
833: L P[833] 240cm/min CNT100 COORD PTH ;
834: L P[834] 240cm/min CNT100 COORD PTH ;
835: L P[835] 240cm/min CNT100 COORD PTH ;
836: L P[836] 240cm/min CNT100 COORD PTH ;
837: L P[837] 240cm/min CNT100 COORD PTH ;
838: L P[838] 240cm/min CNT100 COORD PTH ;
839: L P[839] 240cm/min CNT100 COORD PTH ;
840: L P[840] 240cm/min CNT100 COORD PTH ;
841: L P[841] 240cm/min CNT100 COORD PTH ;
842: L P[842] 240cm/min CNT100 COORD PTH ;
843: L P[843] 240cm/min CNT100 COORD PTH ;
844: L P[844] 240cm/min CNT100 COORD PTH ;
845: L P[845] 240cm/min CNT100 COORD PTH ;
846: L P[846] 240cm/min CNT100 COORD PTH ;
847: L P[847] 240cm/min CNT100 COORD PTH ;
848: L P[848] 240cm/min CNT100 COORD PTH ;
849: L P[849] 240cm/min CNT100 COORD PTH ;
850: L P[850] 240cm/min CNT100 COORD PTH ;
851: L P[851] 240cm/min CNT100 COORD PTH ;
852: L P[852] 240cm/min CNT100 COORD PTH ;
853: L P[853] 240cm/min CNT100 COORD PTH ;
854: L P[854] 240cm/min CNT100 COORD PTH ;
855: L P[855] 240cm/min CNT100 COORD PTH ;
856: L P[856] 240cm/min CNT100 COORD PTH ;
857: L P[857] 240cm/min CNT100 COORD PTH ;
858: L P[858] 240cm/min CNT100 COORD PTH ;
859: L P[859] 240cm/min CNT100 COORD PTH ;
860: L P[860] 240cm/min CNT100 COORD PTH ;
861: L P[861] 240cm/min CNT100 COORD PTH ;
862: L P[862] 240cm/min CNT100 COORD PTH ;
863: L P[863] 240cm/min CNT100 COORD PTH ;
864: L P[864] 240cm/min CNT100 COORD PTH ;
865: L P[865] 240cm/min CNT100 COORD PTH ;
866: L P[866] 240cm/min CNT100 COORD PTH ;
867: L P[867] 240cm/min CNT100 COORD PTH ;
868: L P[868] 240cm/min CNT100 COORD PTH ;
869: L P[869] 240cm/min CNT100 COORD PTH ;
870: L P[870] 240cm/min CNT100 COORD PTH ;
871: L P[871] 240cm/min CNT100 COORD PTH ;
872: L P[872] 240cm/min CNT100 COORD PTH ;
873: L P[873] 240cm/min CNT100 COORD PTH ;
874: L P[874] 240cm/min CNT100 COORD PTH ;
875: L P[875] 240cm/min CNT100 COORD PTH ;
876: L P[876] 240cm/min CNT100 COORD PTH ;
877: L P[877] 240cm/min CNT100 COORD PTH ;
878: L P[878] 240cm/min CNT100 COORD PTH ;
879: L P[879] 240cm/min CNT100 COORD PTH ;
880: L P[880] 240cm/min CNT100 COORD PTH ;
881: L P[881] 240cm/min CNT100 COORD PTH ;
882: L P[882] 240cm/min CNT100 COORD PTH ;
883: L P[883] 240cm/min CNT100 COORD PTH ;
884: L P[884] 240cm/min CNT100 COORD PTH ;
885: L P[885] 240cm/min CNT100 COORD PTH ;
886: L P[886] 240cm/min CNT100 COORD PTH ;
887: L P[887] 240cm/min CNT100 COORD PTH ;
888: L P[888] 240cm/min CNT100 COORD PTH ;
889: L P[889] 240cm/min CNT100 COORD PTH ;
890: L P[890] 240cm/min CNT100 COORD PTH ;
891: L P[891] 240cm/min CNT100 COORD PTH ;
892: L P[892] 240cm/min CNT100 COORD PTH ;
893: L P[893] 240cm/min CNT100 COORD PTH ;
894: L P[894] 240cm/min CNT100 COORD PTH ;
895: L P[895] 240cm/min CNT100 COORD PTH ;
896: L P[896] 240cm/min CNT100 COORD PTH ;
897: L P[897] 240cm/min CNT100 COORD PTH ;
898: L P[898] 240cm/min CNT100 COORD PTH ;
899: L P[899] 240cm/min CNT100 COORD PTH ;
900: L P[900] 240cm/min CNT100 COORD PTH ;
901: L P[901] 240cm/min CNT100 COORD PTH ;
902: L P[902] 240cm/min CNT100 COORD PTH ;
903: L P[903] 240cm/min CNT100 COORD PTH ;
904: L P[904] 240cm/min CNT100 COORD PTH ;
905: L P[905] 240cm/min CNT100 COORD PTH ;
906: L P[906] 240cm/min CNT100 COORD PTH ;
907: L P[907] 240cm/min CNT100 COORD PTH ;
908: L P[908] 240cm/min CNT100 COORD PTH ;
909: L P[909] 240cm/min CNT100 COORD PTH ;
910: L P[910] 240cm/min CNT100 COORD PTH ;
911: L P[911] 240cm/min CNT100 COORD PTH ;
912: L P[912] 240cm/min CNT100 COORD PTH ;
913: L P[913] 240cm/min CNT100 COORD PTH ;
914: L P[914] 240cm/min CNT100 COORD PTH ;
915: L P[915] 240cm/min CNT100 COORD PTH ;
916: L P[916] 240cm/min CNT100 COORD PTH ;
917: L P[917] 240cm/min CNT100 COORD PTH ;
918: L P[918] 240cm/min CNT100 COORD PTH ;
919: L P[919] 240cm/min CNT100 COORD PTH ;
920: L P[920] 240cm/min CNT100 COORD PTH ;
921: L P[921] 240cm/min CNT100 COORD PTH ;
922: L P[922] 240cm/min CNT100 COORD PTH ;
923: L P[923] 240cm/min CNT100 COORD PTH ;
924: L P[924] 240cm/min CNT100 COORD PTH ;
925: L P[925] 240cm/min CNT100 COORD PTH ;
926: L P[926] 240cm/min CNT100 COORD PTH ;
927: L P[927] 240cm/min CNT100 COORD PTH ;
928: L P[928] 240cm/min CNT100 COORD PTH ;
929: L P[929] 240cm/min CNT100 COORD PTH ;
930: L P[930] 240cm/min CNT100 COORD PTH ;
931: L P[931] 240cm/min CNT100 COORD PTH ;
932: L P[932] 240cm/min CNT100 COORD PTH ;
933: L P[933] 240cm/min CNT100 COORD PTH ;
934: L P[934] 240cm/min CNT100 COORD PTH ;
935: L P[935] 240cm/min CNT100 COORD PTH ;
936: L P[936] 240cm/min CNT100 COORD PTH ;
937: L P[937] 240cm/min CNT100 COORD PTH ;
938: L P[938] 240cm/min CNT100 COORD PTH ;
939: L P[939] 240cm/min CNT100 COORD PTH ;
940: L P[940] 240cm/min CNT100 COORD PTH ;
941: L P[941] 240cm/min CNT100 COORD PTH ;
942: L P[942] 240cm/min CNT100 COORD PTH ;
943: L P[943] 240cm/min CNT100 COORD PTH ;
944: L P[944] 240cm/min CNT100 COORD PTH ;
945: L P[945] 240cm/min CNT100 COORD PTH ;
946: L P[946] 240cm/min CNT100 COORD PTH ;
947: L P[947] 240cm/min CNT100 COORD PTH ;
948: L P[948] 240cm/min CNT100 COORD PTH ;
949: L P[949] 240cm/min CNT100 COORD PTH ;
950: L P[950] 240cm/min CNT100 COORD PTH ;
951: L P[951] 240cm/min CNT100 COORD PTH ;
952: L P[952] 240cm/min CNT100 COORD PTH ;
953: L P[953] 240cm/min CNT100 COORD PTH ;
954: L P[954] 240cm/min CNT100 COORD PTH ;
955: L P[955] 240cm/min CNT100 COORD PTH ;
956: L P[956] 240cm/min CNT100 COORD PTH ;
957: L P[957] 240cm/min CNT100 COORD PTH ;
958: L P[958] 240cm/min CNT100 COORD PTH ;
959: L P[959] 240cm/min CNT100 COORD PTH ;
960: L P[960] 240cm/min CNT100 COORD PTH ;
961: L P[961] 240cm/min CNT100 COORD PTH ;
962: L P[962] 240cm/min CNT100 COORD PTH ;
963: L P[963] 240cm/min CNT100 COORD PTH ;
964: L P[964] 240cm/min CNT100 COORD PTH ;
965: L P[965] 240cm/min CNT100 COORD PTH ;
966: L P[966] 240cm/min CNT100 COORD PTH ;
967: L P[967] 240cm/min CNT100 COORD PTH ;
968: L P[968] 240cm/min CNT100 COORD PTH ;
969: L P[969] 240cm/min CNT100 COORD PTH ;
970: L P[970] 240cm/min CNT100 COORD PTH ;
971: L P[971] 240cm/min CNT100 COORD PTH ;
972: L P[972] 240cm/min CNT100 COORD PTH ;
973: L P[973] 240cm/min CNT100 COORD PTH ;
974: L P[974] 240cm/min CNT100 COORD PTH ;
975: L P[975] 240cm/min CNT100 COORD PTH ;
976: L P[976] 240cm/min CNT100 COORD PTH ;
977: L P[977] 240cm/min CNT100 COORD PTH ;
978: L P[978] 240cm/min CNT100 COORD PTH ;
979: L P[979] 240cm/min CNT100 COORD PTH ;
980: L P[980] 240cm/min CNT100 COORD PTH ;
981: L P[981] 240cm/min CNT100 COORD PTH ;
982: L P[982] 240cm/min CNT100 COORD PTH ;
983: L P[983] 240cm/min CNT100 COORD PTH ;
984: L P[984] 240cm/min CNT100 COORD PTH ;
985: L P[985] 240cm/min CNT100 COORD PTH ;
986: L P[986] 240cm/min CNT100 COORD PTH ;
987: L P[987] 240cm/min CNT100 COORD PTH ;
988: L P[988] 240cm/min CNT100 COORD PTH ;
989: L P[989] 240cm/min CNT100 COORD PTH ;
990: L P[990] 240cm/min CNT100 COORD PTH ;
991: L P[991] 240cm/min CNT100 COORD PTH ;
992: L P[992] 240cm/min CNT100 COORD PTH ;
993: L P[993] 240cm/min CNT100 COORD PTH ;
994: L P[994] 240cm/min CNT100 COORD PTH ;
995: L P[995] 240cm/min CNT100 COORD PTH ;
996: L P[996] 240cm/min CNT100 COORD PTH ;
997: L P[997] 240cm/min CNT100 COORD PTH ;
998: L P[998] 240cm/min CNT100 COORD PTH ;
999: L P[999] 240cm/min CNT100 COORD PTH ;
1000: L P[1000] 240cm/min CNT100 COORD PTH ;
1001: L P[1001] 240cm/min CNT100 COORD PTH ;
1002: L P[1002] 240cm/min CNT100 COORD PTH ;
1003: L P[1003] 240cm/min CNT100 COORD PTH ;
1004: L P[1004] 240cm/min CNT100 COORD PTH ;
1005: L P[1005] 240cm/min CNT100 COORD PTH ;
1006: L P[1006] 240cm/min CNT100 COORD PTH ;
1007: L P[1007] 240cm/min CNT100 COORD PTH ;
1008: L P[1008] 240cm/min CNT100 COORD PTH ;
1009: L P[1009] 240cm/min CNT100 COORD PTH ;
1010: L P[1010] 240cm/min CNT100 COORD PTH ;
1011: L P[1011] 240cm/min CNT100 COORD PTH ;
1012: L P[1012] 240cm/min CNT100 COORD PTH ;
1013: L P[1013] 240cm/min CNT100 COORD PTH ;
1014: L P[1014] 240cm/min CNT100 COORD PTH ;
1015: L P[1015] 240cm/min CNT100 COORD PTH ;
1016: L P[1016] 240cm/min CNT100 COORD PTH ;
1017: L P[1017] 240cm/min CNT100 COORD PTH ;
1018: L P[1018] 240cm/min CNT100 COORD PTH ;
1019: L P[1019] 240cm/min CNT100 COORD PTH ;
1020: L P[1020] 240cm/min CNT100 COORD PTH ;
1021: L P[1021] 240cm/min CNT100 COORD PTH ;
1022: L P[1022] 240cm/min CNT100 COORD PTH ;
1023: L P[1023] 240cm/min CNT100 COORD PTH ;
1024: L P[1024] 240cm/min CNT100 COORD PTH ;
1025: L P[1025] 240cm/min CNT100 COORD PTH ;
1026: L P[1026] 240cm/min CNT100 COORD PTH ;
1027: L P[1027] 240cm/min CNT100 COORD PTH ;
1028: L P[1028] 240cm/min CNT100 COORD PTH ;
1029: L P[1029] 240cm/min CNT100 COORD PTH ;
1030: L P[1030] 240cm/min CNT100 COORD PTH ;
1031: L P[1031] 240cm/min CNT100 COORD PTH ;
1032: L P[1032] 240cm/min CNT100 COORD PTH ;
1033: L P[1033] 240cm/min CNT100 COORD PTH ;
1034: L P[1034] 240cm/min CNT100 COORD PTH ;
1035: L P[1035] 240cm/min CNT100 COORD PTH ;
1036: L P[1036] 240cm/min CNT100 COORD PTH ;
1037: L P[1037] 240cm/min CNT100 COORD PTH ;
1038: L P[1038] 240cm/min CNT100 COORD PTH ;
1039: L P[1039] 240cm/min CNT100 COORD PTH ;
1040: L P[1040] 240cm/min CNT100 COORD PTH ;
1041: L P[1041] 240cm/min CNT100 COORD PTH ;
1042: L P[1042] 240cm/min CNT100 COORD PTH ;
1043: L P[1043] 240cm/min CNT100 COORD PTH ;
1044: L P[1044] 240cm/min CNT100 COORD PTH ;
1045: L P[1045] 240cm/min CNT100 COORD PTH ;
1046: L P[1046] 240cm/min CNT100 COORD PTH ;
1047: L P[1047] 240cm/min CNT100 COORD PTH ;
1048: L P[1048] 240cm/min CNT100 COORD PTH ;
1049: L P[1049] 240cm/min CNT100 COORD PTH ;
1050: L P[1050] 240cm/min CNT100 COORD PTH ;
1051: L P[1051] 240cm/min CNT100 COORD PTH ;
1052: L P[1052] 240cm/min CNT100 COORD PTH ;
1053: L P[1053] 240cm/min CNT100 COORD PTH ;
1054: L P[1054] 240cm/min CNT100 COORD PTH ;
1055: L P[1055] 240cm/min CNT100 COORD PTH ;
1056: L P[1056] 240cm/min CNT100 COORD PTH ;
1057: L P[1057] 240cm/min CNT100 COORD PTH ;
1058: L P[1058] 240cm/min CNT100 COORD PTH ;
1059: L P[1059] 240cm/min CNT100 COORD PTH ;
1060: L P[1060] 240cm/min CNT100 COORD PTH ;
1061: L P[1061] 240cm/min CNT100 COORD PTH ;
1062: L P[1062] 240cm/min CNT100 COORD PTH ;
1063: L P[1063] 240cm/min CNT100 COORD PTH ;
1064: L P[1064] 240cm/min CNT100 COORD PTH ;
1065: L P[1065] 240cm/min CNT100 COORD PTH ;
1066: L P[1066] 240cm/min CNT100 COORD PTH ;
1067: L P[1067] 240cm/min CNT100 COORD PTH ;
1068: L P[1068] 240cm/min CNT100 COORD PTH ;
1069: L P[1069] 240cm/min CNT100 COORD PTH ;
1070: L P[1070] 240cm/min CNT100 COORD PTH ;
1071: L P[1071] 240cm/min CNT100 COORD PTH ;
1072: L P[1072] 240cm/min CNT100 COORD PTH ;
1073: L P[1073] 240cm/min CNT100 COORD PTH ;
1074: L P[1074] 240cm/min CNT100 COORD PTH ;
1075: L P[1075] 240cm/min CNT100 COORD PTH ;
1076: L P[1076] 240cm/min CNT100 COORD PTH ;
1077: L P[1077] 240cm/min CNT100 COORD PTH ;
1078: L P[1078] 240cm/min CNT100 COORD PTH ;
1079: L P[1079] 240cm/min CNT100 COORD PTH ;
1080: L P[1080] 240cm/min CNT100 COORD PTH ;
1081: L P[1081] 240cm/min CNT100 COORD PTH ;
1082: L P[1082] 240cm/min CNT100 COORD PTH ;
1083: L P[1083] 240cm/min CNT100 COORD PTH ;
1084: L P[1084] 240cm/min CNT100 COORD PTH ;
1085: L P[1085] 240cm/min CNT100 COORD PTH ;
1086: L P[1086] 240cm/min CNT100 COORD PTH ;
1087: L P[1087] 240cm/min CNT100 COORD PTH ;
1088: L P[1088] 240cm/min CNT100 COORD PTH ;
1089: L P[1089] 240cm/min CNT100 COORD PTH ;
1090: L P[1090] 240cm/min CNT100 COORD PTH ;
1091: L P[1091] 240cm/min CNT100 COORD PTH ;
1092: L P[1092] 240cm/min CNT100 COORD PTH ;
1093: L P[1093] 240cm/min CNT100 COORD PTH ;
1094: L P[1094] 240cm/min CNT100 COORD PTH ;
1095: L P[1095] 240cm/min CNT100 COORD PTH ;
1096: L P[1096] 240cm/min CNT100 COORD PTH ;
1097: L P[1097] 240cm/min CNT100 COORD PTH ;
1098: L P[1098] 240cm/min CNT100 COORD PTH ;
1099: L P[1099] 240cm/min CNT100 COORD PTH ;
1100: L P[1100] 240cm/min CNT100 COORD PTH ;
1101: L P[1101] 240cm/min CNT100 COORD PTH ;
1102: L P[1102] 240cm/min CNT100 COORD PTH ;
1103: L P[1103] 240cm/min CNT100 COORD PTH ;
1104: L P[1104] 240cm/min CNT100 COORD PTH ;
1105: L P[1105] 240cm/min CNT100 COORD PTH ;
1106: L P[1106] 240cm/min CNT100 COORD PTH ;
1107: L P[1107] 240cm/min CNT100 COORD PTH ;
1108: L P[1108] 240cm/min CNT100 COORD PTH ;
1109: L P[1109] 240cm/min CNT100 COORD PTH ;
1110: L P[1110] 240cm/min CNT100 COORD PTH ;
1111: L P[1111] 240cm/min CNT100 COORD PTH ;
1112: L P[1112] 240cm/min CNT100 COORD PTH ;
1113: L P[1113] 240cm/min CNT100 COORD PTH ;
1114: L P[1114] 240cm/min CNT100 COORD PTH ;
1115: L P[1115] 240cm/min CNT100 COORD PTH ;
1116: L P[1116] 240cm/min CNT100 COORD PTH ;
1117: L P[1117] 240cm/min CNT100 COORD PTH ;
1118: L P[1118] 240cm/min CNT100 COORD PTH ;
1119: L P[1119] 240cm/min CNT100 COORD PTH ;
1120: L P[1120] 240cm/min CNT100 COORD PTH ;
1121: L P[1121] 240cm/min CNT100 COORD PTH ;
1122: L P[1122] 240cm/min CNT100 COORD PTH ;
1123: L P[1123] 240cm/min CNT100 COORD PTH ;
1124: L P[1124] 240cm/min CNT100 COORD PTH ;
1125: L P[1125] 240cm/min CNT100 COORD PTH ;
1126: L P[1126] 240cm/min CNT100 COORD PTH ;
1127: L P[1127] 240cm/min CNT100 COORD PTH ;
1128: L P[1128] 240cm/min CNT100 COORD PTH ;
1129: L P[1129] 240cm/min CNT100 COORD PTH ;
1130: L P[1130] 240cm/min CNT100 COORD PTH ;
1131: L P[1131] 240cm/min CNT100 COORD PTH ;
1132: L P[1132] 240cm/min CNT100 COORD PTH ;
1133: L P[1133] 240cm/min CNT100 COORD PTH ;
1134: L P[1134] 240cm/min CNT100 COORD PTH ;
1135: L P[1135] 240cm/min CNT100 COORD PTH ;
1136: L P[1136] 240cm/min CNT100 COORD PTH ;
1137: L P[1137] 240cm/min CNT100 COORD PTH ;
1138: L P[1138] 240cm/min CNT100 COORD PTH ;
1139: L P[1139] 240cm/min CNT100 COORD PTH ;
1140: L P[1140] 240cm/min CNT100 COORD PTH ;
1141: L P[1141] 240cm/min CNT100 COORD PTH ;
1142: L P[1142] 240cm/min CNT100 COORD PTH ;
1143: L P[1143] 240cm/min CNT100 COORD PTH ;
1144: L P[1144] 240cm/min CNT100 COORD PTH ;
1145: L P[1145] 240cm/min CNT100 COORD PTH ;
1146: L P[1146] 240cm/min CNT100 COORD PTH ;
1147: L P[1147] 240cm/min CNT100 COORD PTH ;
1148: L P[1148] 240cm/min CNT100 COORD PTH ;
1149: L P[1149] 240cm/min CNT100 COORD PTH ;
1150: L P[1150] 240cm/min CNT100 COORD PTH ;
1151: L P[1151] 240cm/min CNT100 COORD PTH ;
1152: L P[1152] 240cm/min CNT100 COORD PTH ;
1153: L P[1153] 240cm/min CNT100 COORD PTH ;
1154: L P[1154] 240cm/min CNT100 COORD PTH ;
1155: L P[1155] 240cm/min CNT100 COORD PTH ;
1156: L P[1156] 240cm/min CNT100 COORD PTH ;
1157: L P[1157] 240cm/min CNT100 COORD PTH ;
1158: L P[1158] 240cm/min CNT100 COORD PTH ;
1159: L P[1159] 240cm/min CNT100 COORD PTH ;
1160: L P[1160] 240cm/min CNT100 COORD PTH ;
1161: L P[1161] 240cm/min CNT100 COORD PTH ;
1162: L P[1162] 240cm/min CNT100 COORD PTH ;
1163: L P[1163] 240cm/min CNT100 COORD PTH ;
1164: L P[1164] 240cm/min CNT100 COORD PTH ;
1165: L P[1165] 240cm/min CNT100 COORD PTH ;
1166: L P[1166] 240cm/min CNT100 COORD PTH ;
1167: L P[1167] 240cm/min CNT100 COORD PTH ;
1168: L P[1168] 240cm/min CNT100 COORD PTH ;
1169: L P[1169] 240cm/min CNT100 COORD PTH ;
1170: L P[1170] 240cm/min CNT100 COORD PTH ;
1171: L P[1171] 240cm/min CNT100 COORD PTH ;
1172: L P[1172] 240cm/min CNT100 COORD PTH ;
1173: L P[1173] 240cm/min CNT100 COORD PTH ;
1174: L P[1174] 240cm/min CNT100 COORD PTH ;
1175: L P[1175] 240cm/min CNT100 COORD PTH ;
1176: L P[1176] 240cm/min CNT100 COORD PTH ;
1177: L P[1177] 240cm/min CNT100 COORD PTH ;
1178: L P[1178] 240cm/min CNT100 COORD PTH ;
1179: L P[1179] 240cm/min CNT100 COORD PTH ;
1180: L P[1180] 240cm/min CNT100 COORD PTH ;
1181: L P[1181] 240cm/min CNT100 COORD PTH ;
1182: L P[1182] 240cm/min CNT100 COORD PTH ;
1183: L P[1183] 240cm/min CNT100 COORD PTH ;
1184: L P[1184] 240cm/min CNT100 COORD PTH ;
1185: L P[1185] 240cm/min CNT100 COORD PTH ;
1186: L P[1186] 240cm/min CNT100 COORD PTH ;
1187: L P[1187] 240cm/min CNT100 COORD PTH ;
1188: L P[1188] 240cm/min CNT100 COORD PTH ;
1189: L P[1189] 240cm/min CNT100 COORD PTH ;
1190: L P[1190] 240cm/min CNT100 COORD PTH ;
1191: L P[1191] 240cm/min CNT100 COORD PTH ;
1192: L P[1192] 240cm/min CNT100 COORD PTH ;
1193: L P[1193] 240cm/min CNT100 COORD PTH ;
1194: L P[1194] 240cm/min CNT100 COORD PTH ;
1195: L P[1195] 240cm/min CNT100 COORD PTH ;
1196: L P[1196] 240cm/min CNT100 COORD PTH ;
1197: L P[1197] 240cm/min CNT100 COORD PTH ;
1198: L P[1198] 240cm/min CNT100 COORD PTH ;
1199: L P[1199] 240cm/min CNT100 COORD PTH ;
1200: L P[1200] 240cm/min CNT100 COORD PTH ;
1201: L P[1201] 240cm/min CNT100 COORD PTH ;
1202: L P[1202] 240cm/min CNT100 COORD PTH ;
1203: L P[1203] 240cm/min CNT100 COORD PTH ;
1204: L P[1204] 240cm/min CNT100 COORD PTH ;
1205: L P[1205] 240cm/min CNT100 COORD PTH ;
1206: L P[1206] 240cm/min CNT100 COORD PTH ;
1207: L P[1207] 240cm/min CNT100 COORD PTH ;
1208: L P[1208] 240cm/min CNT100 COORD PTH ;
1209: L P[1209] 240cm/min CNT100 COORD PTH ;
1210: L P[1210] 240cm/min CNT100 COORD PTH ;
1211: L P[1211] 240cm/min CNT100 COORD PTH ;
1212: L P[1212] 240cm/min CNT100 COORD PTH ;
1213: L P[1213] 240cm/min CNT100 COORD PTH ;
1214: L P[1214] 240cm/min CNT100 COORD PTH ;
1215: L P[1215] 240cm/min CNT100 COORD PTH ;
1216: L P[1216] 240cm/min CNT100 COORD PTH ;
1217: L P[1217] 240cm/min CNT100 COORD PTH ;
1218: L P[1218] 240cm/min CNT100 COORD PTH ;
1219: L P[1219] 240cm/min CNT100 COORD PTH ;
1220: L P[1220] 240cm/min CNT100 COORD PTH ;
1221: L P[1221] 240cm/min CNT100 COORD PTH ;
1222: L P[1222] 240cm/min CNT100 COORD PTH ;
1223: L P[1223] 240cm/min CNT100 COORD PTH ;
1224: L P[1224] 240cm/min CNT100 COORD PTH ;
1225: L P[1225] 240cm/min CNT100 COORD PTH ;
1226: L P[1226] 240cm/min CNT100 COORD PTH ;
1227: L P[1227] 240cm/min CNT100 COORD PTH ;
1228: L P[1228] 240cm/min CNT100 COORD PTH ;
1229: L P[1229] 240cm/min CNT100 COORD PTH ;
1230: L P[1230] 240cm/min CNT100 COORD PTH ;
1231: L P[1231] 240cm/min CNT100 COORD PTH ;
1232: L P[1232] 240cm/min CNT100 COORD PTH ;
1233: L P[1233] 240cm/min CNT100 COORD PTH ;
1234: L P[1234] 240cm/min CNT100 COORD PTH ;
1235: L P[1235] 240cm/min CNT100 COORD PTH ;
1236: L P[1236] 240cm/min CNT100 COORD PTH ;
1237: L P[1237] 240cm/min CNT100 COORD PTH ;
1238: L P[1238] 240cm/min CNT100 COORD PTH ;
1239: L P[1239] 240cm/min CNT100 COORD PTH ;
1240: L P[1240] 240cm/min CNT100 COORD PTH ;
1241: L P[1241] 240cm/min CNT100 COORD PTH ;
1242: L P[1242] 240cm/min CNT100 COORD PTH ;
1243: L P[1243] 240cm/min CNT100 COORD PTH ;
1244: L P[1244] 240cm/min CNT100 COORD PTH ;
1245: L P[1245] 240cm/min CNT100 COORD PTH ;
1246: L P[1246] 240cm/min CNT100 COORD PTH ;
1247: L P[1247] 240cm/min CNT100 COORD PTH ;
1248: L P[1248] 240cm/min CNT100 COORD PTH ;
1249: L P[1249] 240cm/min CNT100 COORD PTH ;
1250: L P[1250] 240cm/min CNT100 COORD PTH ;
1251: L P[1251] 240cm/min CNT100 COORD PTH ;
1252: L P[1252] 240cm/min CNT100 COORD PTH ;
1253: L P[1253] 240cm/min CNT100 COORD PTH ;
1254: L P[1254] 240cm/min CNT100 COORD PTH ;
1255: L P[1255] 240cm/min CNT100 COORD PTH ;
1256: L P[1256] 240cm/min CNT100 COORD PTH ;
1257: L P[1257] 240cm/min CNT100 COORD PTH ;
1258: L P[1258] 240cm/min CNT100 COORD PTH ;
1259: L P[1259] 240cm/min CNT100 COORD PTH ;
1260: L P[1260] 240cm/min CNT100 COORD PTH ;
1261: L P[1261] 240cm/min CNT100 COORD PTH ;
1262: L P[1262] 240cm/min CNT100 COORD PTH ;
1263: L P[1263] 240cm/min CNT100 COORD PTH ;
1264: L P[1264] 240cm/min CNT100 COORD PTH ;
1265: L P[1265] 240cm/min CNT100 COORD PTH ;
1266: L P[1266] 240cm/min CNT100 COORD PTH ;
1267: L P[1267] 240cm/min CNT100 COORD PTH ;
1268: L P[1268] 240cm/min CNT100 COORD PTH ;
1269: L P[1269] 240cm/min CNT100 COORD PTH ;
1270: L P[1270] 240cm/min CNT100 COORD PTH ;
1271: L P[1271] 240cm/min CNT100 COORD PTH ;
1272: L P[1272] 240cm/min CNT100 COORD PTH ;
1273: L P[1273] 240cm/min CNT100 COORD PTH ;
1274: L P[1274] 240cm/min CNT100 COORD PTH ;
1275: L P[1275] 240cm/min CNT100 COORD PTH ;
1276: L P[1276] 240cm/min CNT100 COORD PTH ;
1277: L P[1277] 240cm/min CNT100 COORD PTH ;
1278: L P[1278] 240cm/min CNT100 COORD PTH ;
1279: L P[1279] 240cm/min CNT100 COORD PTH ;
1280: L P[1280] 240cm/min CNT100 COORD PTH ;
1281: L P[1281] 240cm/min CNT100 COORD PTH ;
1282: L P[1282] 240cm/min CNT100 COORD PTH ;
1283: L P[1283] 240cm/min CNT100 COORD PTH ;
1284: L P[1284] 240cm/min CNT100 COORD PTH ;
1285: L P[1285] 240cm/min CNT100 COORD PTH ;
1286: L P[1286] 240cm/min CNT100 COORD PTH ;
1287: L P[1287] 240cm/min CNT100 COORD PTH ;
1288: L P[1288] 240cm/min CNT100 COORD PTH ;
1289: L P[1289] 240cm/min CNT100 COORD PTH ;
1290: L P[1290] 240cm/min CNT100 COORD PTH ;
1291: L P[1291] 240cm/min CNT100 COORD PTH ;
1292: L P[1292] 240cm/min CNT100 COORD PTH ;
1293: L P[1293] 240cm/min CNT100 COORD PTH ;
1294: L P[1294] 240cm/min CNT100 COORD PTH ;
1295: L P[1295] 240cm/min CNT100 COORD PTH ;
1296: L P[1296] 240cm/min CNT100 COORD PTH ;
1297: L P[1297] 240cm/min CNT100 COORD PTH ;
1298: L P[1298] 240cm/min CNT100 COORD PTH ;
1299: L P[1299] 240cm/min CNT100 COORD PTH ;
1300: L P[1300] 240cm/min CNT100 COORD PTH ;
1301: L P[1301] 240cm/min CNT100 COORD PTH ;
1302: L P[1302] 240cm/min CNT100 COORD PTH ;
1303: L P[1303] 240cm/min CNT100 COORD PTH ;
1304: L P[1304] 240cm/min CNT100 COORD PTH ;
1305: L P[1305] 240cm/min CNT100 COORD PTH ;
1306: L P[1306] 240cm/min CNT100 COORD PTH ;
1307: L P[1307] 240cm/min CNT100 COORD PTH ;
1308: L P[1308] 240cm/min CNT100 COORD PTH ;
1309: L P[1309] 240cm/min CNT100 COORD PTH ;
1310: L P[1310] 240cm/min CNT100 COORD PTH ;
1311: L P[1311] 240cm/min CNT100 COORD PTH ;
1312: L P[1312] 240cm/min CNT100 COORD PTH ;
1313: L P[1313] 240cm/min CNT100 COORD PTH ;
1314: L P[1314] 240cm/min CNT100 COORD PTH ;
1315: L P[1315] 240cm/min CNT100 COORD PTH ;
1316: L P[1316] 240cm/min CNT100 COORD PTH ;
1317: L P[1317] 240cm/min CNT100 COORD PTH ;
1318: L P[1318] 240cm/min CNT100 COORD PTH ;
1319: L P[1319] 240cm/min CNT100 COORD PTH ;
1320: L P[1320] 240cm/min CNT100 COORD PTH ;
1321: L P[1321] 240cm/min CNT100 COORD PTH ;
1322: L P[1322] 240cm/min CNT100 COORD PTH ;
1323: L P[1323] 240cm/min CNT100 COORD PTH ;
1324: L P[1324] 240cm/min CNT100 COORD PTH ;
1325: L P[1325] 240cm/min CNT100 COORD PTH ;
1326: L P[1326] 240cm/min CNT100 COORD PTH ;
1327: L P[1327] 240cm/min CNT100 COORD PTH ;
1328: L P[1328] 240cm/min CNT100 COORD PTH ;
1329: L P[1329] 240cm/min CNT100 COORD PTH ;
1330: L P[1330] 240cm/min CNT100 COORD PTH ;
1331: L P[1331] 240cm/min CNT100 COORD PTH ;
1332: L P[1332] 240cm/min CNT100 COORD PTH ;
1333: L P[1333] 240cm/min CNT100 COORD PTH ;
1334: L P[1334] 240cm/min CNT100 COORD PTH ;
1335: L P[1335] 240cm/min CNT100 COORD PTH ;
1336: L P[1336] 240cm/min CNT100 COORD PTH ;
1337: L P[1337] 240cm/min CNT100 COORD PTH ;
1338: L P[1338] 240cm/min CNT100 COORD PTH ;
1339: L P[1339] 240cm/min CNT100 COORD PTH ;
1340: L P[1340] 240cm/min CNT100 COORD PTH ;
1341: L P[1341] 240cm/min CNT100 COORD PTH ;
1342: L P[1342] 240cm/min CNT100 COORD PTH ;
1343: L P[1343] 240cm/min CNT100 COORD PTH ;
1344: L P[1344] 240cm/min CNT100 COORD PTH ;
1345: L P[1345] 240cm/min CNT100 COORD PTH ;
1346: L P[1346] 240cm/min CNT100 COORD PTH ;
1347: L P[1347] 240cm/min CNT100 COORD PTH ;
1348: L P[1348] 240cm/min CNT100 COORD PTH ;
1349: L P[1349] 240cm/min CNT100 COORD PTH ;
1350: L P[1350] 240cm/min CNT100 COORD PTH ;
1351: L P[1351] 240cm/min CNT100 COORD PTH ;
1352: L P[1352] 240cm/min CNT100 COORD PTH ;
1353: L P[1353] 240cm/min CNT100 COORD PTH ;
1354: L P[1354] 240cm/min CNT100 COORD PTH ;
1355: L P[1355] 240cm/min CNT100 COORD PTH ;
1356: L P[1356] 240cm/min CNT100 COORD PTH ;
1357: L P[1357] 240cm/min CNT100 COORD PTH ;
1358: L P[1358] 240cm/min CNT100 COORD PTH ;
1359: L P[1359] 240cm/min CNT100 COORD PTH ;
1360: L P[1360] 240cm/min CNT100 COORD PTH ;
1361: L P[1361] 240cm/min CNT100 COORD PTH ;
1362: L P[1362] 240cm/min CNT100 COORD PTH ;
1363: L P[1363] 240cm/min CNT100 COORD PTH ;
1364: L P[1364] 240cm/min CNT100 COORD PTH ;
1365: L P[1365] 240cm/min CNT100 COORD PTH ;
1366: L P[1366] 240cm/min CNT100 COORD PTH ;
1367: L P[1367] 240cm/min CNT100 COORD PTH ;
1368: L P[1368] 240cm/min CNT100 COORD PTH ;
1369: L P[1369] 240cm/min CNT100 COORD PTH ;
1370: L P[1370] 240cm/min CNT100 COORD PTH ;
1371: L P[1371] 240cm/min CNT100 COORD PTH ;
1372: L P[1372] 240cm/min CNT100 COORD PTH ;
1373: L P[1373] 240cm/min CNT100 COORD PTH ;
1374: L P[1374] 240cm/min CNT100 COORD PTH ;
1375: L P[1375] 240cm/min CNT100 COORD PTH ;
1376: L P[1376] 240cm/min CNT100 COORD PTH ;
1377: L P[1377] 240cm/min CNT100 COORD PTH ;
1378: L P[1378] 240cm/min CNT100 COORD PTH ;
1379: L P[1379] 240cm/min CNT100 COORD PTH ;
1380: L P[1380] 240cm/min CNT100 COORD PTH ;
1381: L P[1381] 240cm/min CNT100 COORD PTH ;
1382: L P[1382] 240cm/min CNT100 COORD PTH ;
1383: L P[1383] 240cm/min CNT100 COORD PTH ;
1384: L P[1384] 240cm/min CNT100 COORD PTH ;
1385: L P[1385] 240cm/min CNT100 COORD PTH ;
1386: L P[1386] 240cm/min CNT100 COORD PTH ;
1387: L P[1387] 240cm/min CNT100 COORD PTH ;
1388: L P[1388] 240cm/min CNT100 COORD PTH ;
1389: L P[1389] 240cm/min CNT100 COORD PTH ;
1390: L P[1390] 240cm/min CNT100 COORD PTH ;
1391: L P[1391] 240cm/min CNT100 COORD PTH ;
1392: L P[1392] 240cm/min CNT100 COORD PTH ;
1393: L P[1393] 240cm/min CNT100 COORD PTH ;
1394: L P[1394] 240cm/min CNT100 COORD PTH ;
1395: L P[1395] 240cm/min CNT100 COORD PTH ;
1396: L P[1396] 240cm/min CNT100 COORD PTH ;
1397: L P[1397] 240cm/min CNT100 COORD PTH ;
1398: L P[1398] 240cm/min CNT100 COORD PTH ;
1399: L P[1399] 240cm/min CNT100 COORD PTH ;
1400: L P[1400] 240cm/min CNT100 COORD PTH ;
1401: L P[1401] 240cm/min CNT100 COORD PTH ;
1402: L P[1402] 240cm/min CNT100 COORD PTH ;
1403: L P[1403] 240cm/min CNT100 COORD PTH ;
1404: L P[1404] 240cm/min CNT100 COORD PTH ;
1405: L P[1405] 240cm/min CNT100 COORD PTH ;
1406: L P[1406] 240cm/min CNT100 COORD PTH ;
1407: L P[1407] 240cm/min CNT100 COORD PTH ;
1408: L P[1408] 240cm/min CNT100 COORD PTH ;
1409: L P[1409] 240cm/min CNT100 COORD PTH ;
1410: L P[1410] 240cm/min CNT100 COORD PTH ;
1411: L P[1411] 240cm/min CNT100 COORD PTH ;
1412: L P[1412] 240cm/min CNT100 COORD PTH ;
1413: L P[1413] 240cm/min CNT100 COORD PTH ;
1414: L P[1414] 240cm/min CNT100 COORD PTH ;
1415: L P[1415] 240cm/min CNT100 COORD PTH ;
1416: L P[1416] 240cm/min CNT100 COORD PTH ;
1417: L P[1417] 240cm/min CNT100 COORD PTH ;
1418: L P[1418] 240cm/min CNT100 COORD PTH ;
1419: L P[1419] 240cm/min CNT100 COORD PTH ;
1420: L P[1420] 240cm/min CNT100 COORD PTH ;
1421: L P[1421] 240cm/min CNT100 COORD PTH ;
1422: L P[1422] 240cm/min CNT100 COORD PTH ;
1423: L P[1423] 240cm/min CNT100 COORD PTH ;
1424: L P[1424] 240cm/min CNT100 COORD PTH ;
1425: L P[1425] 240cm/min CNT100 COORD PTH ;
1426: L P[1426] 240cm/min CNT100 COORD PTH ;
1427: L P[1427] 240cm/min CNT100 COORD PTH ;
1428: L P[1428] 240cm/min CNT100 COORD PTH ;
1429: L P[1429] 240cm/min CNT100 COORD PTH ;
1430: L P[1430] 240cm/min CNT100 COORD PTH ;
1431: L P[1431] 240cm/min CNT100 COORD PTH ;
1432: L P[1432] 240cm/min CNT100 COORD PTH ;
1433: L P[1433] 240cm/min CNT100 COORD PTH ;
1434: L P[1434] 240cm/min CNT100 COORD PTH ;
1435: L P[1435] 240cm/min CNT100 COORD PTH ;
1436: L P[1436] 240cm/min CNT100 COORD PTH ;
1437: L P[1437] 240cm/min CNT100 COORD PTH ;
1438: L P[1438] 240cm/min CNT100 COORD PTH ;
1439: L P[1439] 240cm/min CNT100 COORD PTH ;
1440: L P[1440] 240cm/min CNT100 COORD PTH ;
1441: L P[1441] 240cm/min CNT100 COORD PTH ;
1442: L P[1442] 240cm/min CNT100 COORD PTH ;
1443: L P[1443] 240cm/min CNT100 COORD PTH ;
1444: L P[1444] 240cm/min CNT100 COORD PTH ;
1445: L P[1445] 240cm/min CNT100 COORD PTH ;
1446: L P[1446] 240cm/min CNT100 COORD PTH ;
1447: L P[1447] 240cm/min CNT100 COORD PTH ;
1448: L P[1448] 240cm/min CNT100 COORD PTH ;
1449: L P[1449] 240cm/min CNT100 COORD PTH ;
1450: L P[1450] 240cm/min CNT100 COORD PTH ;
1451: L P[1451] 240cm/min CNT100 COORD PTH ;
1452: L P[1452] 240cm/min CNT100 COORD PTH ;
1453: L P[1453] 240cm/min CNT100 COORD PTH ;
1454: L P[1454] 240cm/min CNT100 COORD PTH ;
1455: L P[1455] 240cm/min CNT100 COORD PTH ;
1456: L P[1456] 240cm/min CNT100 COORD PTH ;
1457: L P[1457] 240cm/min CNT100 COORD PTH ;
1458: L P[1458] 240cm/min CNT100 COORD PTH ;
1459: L P[1459] 240cm/min CNT100 COORD PTH ;
1460: L P[1460] 240cm/min CNT100 COORD PTH ;
1461: L P[1461] 240cm/min CNT100 COORD PTH ;
1462: L P[1462] 240cm/min CNT100 COORD PTH ;
1463: L P[1463] 240cm/min CNT100 COORD PTH ;
1464: L P[1464] 240cm/min CNT100 COORD PTH ;
1465: L P[1465] 240cm/min CNT100 COORD PTH ;
1466: L P[1466] 240cm/min CNT100 COORD PTH ;
1467: L P[1467] 240cm/min CNT100 COORD PTH ;
1468: L P[1468] 240cm/min CNT100 COORD PTH ;
1469: L P[1469] 240cm/min CNT100 COORD PTH ;
1470: L P[1470] 240cm/min CNT100 COORD PTH ;
1471: L P[1471] 240cm/min CNT100 COORD PTH ;
1472: L P[1472] 240cm/min CNT100 COORD PTH ;
1473: L P[1473] 240cm/min CNT100 COORD PTH ;
1474: L P[1474] 240cm/min CNT100 COORD PTH ;
1475: L P[1475] 240cm/min CNT100 COORD PTH ;
1476: L P[1476] 240cm/min CNT100 COORD PTH ;
1477: L P[1477] 240cm/min CNT100 COORD PTH ;
1478: L P[1478] 240cm/min CNT100 COORD PTH ;
1479: L P[1479] 240cm/min CNT100 COORD PTH ;
1480: L P[1480] 240cm/min CNT100 COORD PTH ;
1481: L P[1481] 240cm/min CNT100 COORD PTH ;
1482: L P[1482] 240cm/min CNT100 COORD PTH ;
1483: L P[1483] 240cm/min CNT100 COORD PTH ;
1484: L P[1484] 240cm/min CNT100 COORD PTH ;
1485: L P[1485] 240cm/min CNT100 COORD PTH ;
1486: L P[1486] 240cm/min CNT100 COORD PTH ;
1487: L P[1487] 240cm/min CNT100 COORD PTH ;
1488: L P[1488] 240cm/min CNT100 COORD PTH ;
1489: L P[1489] 240cm/min CNT100 COORD PTH ;
1490: L P[1490] 240cm/min CNT100 COORD PTH ;
1491: L P[1491] 240cm/min CNT100 COORD PTH ;
1492: L P[1492] 240cm/min CNT100 COORD PTH ;
1493: L P[1493] 240cm/min CNT100 COORD PTH ;
1494: L P[1494] 240cm/min CNT100 COORD PTH ;
1495: L P[1495] 240cm/min CNT100 COORD PTH ;
1496: L P[1496] 240cm/min CNT100 COORD PTH ;
1497: L P[1497] 240cm/min CNT100 COORD PTH ;
1498: L P[1498] 240cm/min CNT100 COORD PTH ;
1499: L P[1499] 240cm/min CNT100 COORD PTH ;
1500: L P[1500] 240cm/min CNT100 COORD PTH ;
1501: L P[1501] 240cm/min CNT100 COORD PTH ;
1502: L P[1502] 240cm/min CNT100 COORD PTH ;
1503: L P[1503] 240cm/min CNT100 COORD PTH ;
1504: L P[1504] 240cm/min CNT100 COORD PTH ;
1505: L P[1505] 240cm/min CNT100 COORD PTH ;
1506: L P[1506] 240cm/min CNT100 COORD PTH ;
1507: L P[1507] 240cm/min CNT100 COORD PTH ;
1508: L P[1508] 240cm/min CNT100 COORD PTH ;
1509: L P[1509] 240cm/min CNT100 COORD PTH ;
1510: L P[1510] 240cm/min CNT100 COORD PTH ;
1511: L P[1511] 240cm/min CNT100 COORD PTH ;
1512: L P[1512] 240cm/min CNT100 COORD PTH ;
1513: L P[1513] 240cm/min CNT100 COORD PTH ;
1514: L P[1514] 240cm/min CNT100 COORD PTH ;
1515: L P[1515] 240cm/min CNT100 COORD PTH ;
1516: L P[1516] 240cm/min CNT100 COORD PTH ;
1517: L P[1517] 240cm/min CNT100 COORD PTH ;
1518: L P[1518] 240cm/min CNT100 COORD PTH ;
1519: L P[1519] 240cm/min CNT100 COORD PTH ;
1520: L P[1520] 240cm/min CNT100 COORD PTH ;
1521: L P[1521] 240cm/min CNT100 COORD PTH ;
1522: L P[1522] 240cm/min CNT100 COORD PTH ;
1523: L P[1523] 240cm/min CNT100 COORD PTH ;
1524: L P[1524] 240cm/min CNT100 COORD PTH ;
1525: L P[1525] 240cm/min CNT100 COORD PTH ;
1526: L P[1526] 240cm/min CNT100 COORD PTH ;
1527: L P[1527] 240cm/min CNT100 COORD PTH ;
1528: L P[1528] 240cm/min CNT100 COORD PTH ;
1529: L P[1529] 240cm/min CNT100 COORD PTH ;
1530: L P[1530] 240cm/min CNT100 COORD PTH ;
1531: L P[1531] 240cm/min CNT100 COORD PTH ;
1532: L P[1532] 240cm/min CNT100 COORD PTH ;
1533: L P[1533] 240cm/min CNT100 COORD PTH ;
1534: L P[1534] 240cm/min CNT100 COORD PTH ;
1535: L P[1535] 240cm/min CNT100 COORD PTH ;
1536: L P[1536] 240cm/min CNT100 COORD PTH ;
1537: L P[1537] 240cm/min CNT100 COORD PTH ;
1538: L P[1538] 240cm/min CNT100 COORD PTH ;
1539: L P[1539] 240cm/min CNT100 COORD PTH ;
1540: L P[1540] 240cm/min CNT100 COORD PTH ;
1541: L P[1541] 240cm/min CNT100 COORD PTH ;
1542: L P[1542] 240cm/min CNT100 COORD PTH ;
1543: L P[1543] 240cm/min CNT100 COORD PTH ;
1544: L P[1544] 240cm/min CNT100 COORD PTH ;
1545: L P[1545] 240cm/min CNT100 COORD PTH ;
1546: L P[1546] 240cm/min CNT100 COORD PTH ;
1547: L P[1547] 240cm/min CNT100 COORD PTH ;
1548: L P[1548] 240cm/min CNT100 COORD PTH ;
1549: L P[1549] 240cm/min CNT100 COORD PTH ;
1550: L P[1550] 240cm/min CNT100 COORD PTH ;
1551: L P[1551] 240cm/min CNT100 COORD PTH ;
1552: L P[1552] 240cm/min CNT100 COORD PTH ;
1553: L P[1553] 240cm/min CNT100 COORD PTH ;
1554: L P[1554] 240cm/min CNT100 COORD PTH ;
1555: L P[1555] 240cm/min CNT100 COORD PTH ;
1556: L P[1556] 240cm/min CNT100 COORD PTH ;
1557: L P[1557] 240cm/min CNT100 COORD PTH ;
1558: L P[1558] 240cm/min CNT100 COORD PTH ;
1559: L P[1559] 240cm/min CNT100 COORD PTH ;
1560: L P[1560] 240cm/min CNT100 COORD PTH ;
1561: L P[1561] 240cm/min CNT100 COORD PTH ;
1562: L P[1562] 240cm/min CNT100 COORD PTH ;
1563: L P[1563] 240cm/min CNT100 COORD PTH ;
1564: L P[1564] 240cm/min CNT100 COORD PTH ;
1565: L P[1565] 240cm/min CNT100 COORD PTH ;
1566: L P[1566] 240cm/min CNT100 COORD PTH ;
1567: L P[1567] 240cm/min CNT100 COORD PTH ;
1568: L P[1568] 240cm/min CNT100 COORD PTH ;
1569: L P[1569] 240cm/min CNT100 COORD PTH ;
1570: L P[1570] 240cm/min CNT100 COORD PTH ;
1571: L P[1571] 240cm/min CNT100 COORD PTH ;
1572: L P[1572] 240cm/min CNT100 COORD PTH ;
1573: L P[1573] 240cm/min CNT100 COORD PTH ;
1574: L P[1574] 240cm/min CNT100 COORD PTH ;
1575: L P[1575] 240cm/min CNT100 COORD PTH ;
1576: L P[1576] 240cm/min CNT100 COORD PTH ;
1577: L P[1577] 240cm/min CNT100 COORD PTH ;
1578: L P[1578] 240cm/min CNT100 COORD PTH ;
1579: L P[1579] 240cm/min CNT100 COORD PTH ;
1580: L P[1580] 240cm/min CNT100 COORD PTH ;
1581: L P[1581] 240cm/min CNT100 COORD PTH ;
1582: L P[1582] 240cm/min CNT100 COORD PTH ;
1583: L P[1583] 240cm/min CNT100 COORD PTH ;
1584: L P[1584] 240cm/min CNT100 COORD PTH ;
: Arc End[1];
1585: L P[1585] 240cm/min CNT100 COORD ;
: Arc Start[1];
1586: L P[1586] 240cm/min CNT100 COORD PTH ;
1587: L P[1587] 240cm/min CNT100 COORD PTH ;
1588: L P[1588] 240cm/min CNT100 COORD PTH ;
1589: L P[1589] 240cm/min CNT100 COORD PTH ;
1590: L P[1590] 240cm/min CNT100 COORD PTH ;
1591: L P[1591] 240cm/min CNT100 COORD PTH ;
1592: L P[1592] 240cm/min CNT100 COORD PTH ;
1593: L P[1593] 240cm/min CNT100 COORD PTH ;
1594: L P[1594] 240cm/min CNT100 COORD PTH ;
1595: L P[1595] 240cm/min CNT100 COORD PTH ;
1596: L P[1596] 240cm/min CNT100 COORD PTH ;
1597: L P[1597] 240cm/min CNT100 COORD PTH ;
1598: L P[1598] 240cm/min CNT100 COORD PTH ;
1599: L P[1599] 240cm/min CNT100 COORD PTH ;
1600: L P[1600] 240cm/min CNT100 COORD PTH ;
1601: L P[1601] 240cm/min CNT100 COORD PTH ;
1602: L P[1602] 240cm/min CNT100 COORD PTH ;
1603: L P[1603] 240cm/min CNT100 COORD PTH ;
1604: L P[1604] 240cm/min CNT100 COORD PTH ;
1605: L P[1605] 240cm/min CNT100 COORD PTH ;
1606: L P[1606] 240cm/min CNT100 COORD PTH ;
1607: L P[1607] 240cm/min CNT100 COORD PTH ;
1608: L P[1608] 240cm/min CNT100 COORD PTH ;
1609: L P[1609] 240cm/min CNT100 COORD PTH ;
1610: L P[1610] 240cm/min CNT100 COORD PTH ;
1611: L P[1611] 240cm/min CNT100 COORD PTH ;
1612: L P[1612] 240cm/min CNT100 COORD PTH ;
1613: L P[1613] 240cm/min CNT100 COORD PTH ;
1614: L P[1614] 240cm/min CNT100 COORD PTH ;
1615: L P[1615] 240cm/min CNT100 COORD PTH ;
1616: L P[1616] 240cm/min CNT100 COORD PTH ;
1617: L P[1617] 240cm/min CNT100 COORD PTH ;
1618: L P[1618] 240cm/min CNT100 COORD PTH ;
1619: L P[1619] 240cm/min CNT100 COORD PTH ;
1620: L P[1620] 240cm/min CNT100 COORD PTH ;
1621: L P[1621] 240cm/min CNT100 COORD PTH ;
1622: L P[1622] 240cm/min CNT100 COORD PTH ;
1623: L P[1623] 240cm/min CNT100 COORD PTH ;
1624: L P[1624] 240cm/min CNT100 COORD PTH ;
1625: L P[1625] 240cm/min CNT100 COORD PTH ;
1626: L P[1626] 240cm/min CNT100 COORD PTH ;
1627: L P[1627] 240cm/min CNT100 COORD PTH ;
1628: L P[1628] 240cm/min CNT100 COORD PTH ;
1629: L P[1629] 240cm/min CNT100 COORD PTH ;
1630: L P[1630] 240cm/min CNT100 COORD PTH ;
1631: L P[1631] 240cm/min CNT100 COORD PTH ;
1632: L P[1632] 240cm/min CNT100 COORD PTH ;
1633: L P[1633] 240cm/min CNT100 COORD PTH ;
1634: L P[1634] 240cm/min CNT100 COORD PTH ;
1635: L P[1635] 240cm/min CNT100 COORD PTH ;
1636: L P[1636] 240cm/min CNT100 COORD PTH ;
1637: L P[1637] 240cm/min CNT100 COORD PTH ;
1638: L P[1638] 240cm/min CNT100 COORD PTH ;
1639: L P[1639] 240cm/min CNT100 COORD PTH ;
1640: L P[1640] 240cm/min CNT100 COORD PTH ;
1641: L P[1641] 240cm/min CNT100 COORD PTH ;
1642: L P[1642] 240cm/min CNT100 COORD PTH ;
1643: L P[1643] 240cm/min CNT100 COORD PTH ;
1644: L P[1644] 240cm/min CNT100 COORD PTH ;
1645: L P[1645] 240cm/min CNT100 COORD PTH ;
1646: L P[1646] 240cm/min CNT100 COORD PTH ;
1647: L P[1647] 240cm/min CNT100 COORD PTH ;
1648: L P[1648] 240cm/min CNT100 COORD PTH ;
1649: L P[1649] 240cm/min CNT100 COORD PTH ;
1650: L P[1650] 240cm/min CNT100 COORD PTH ;
1651: L P[1651] 240cm/min CNT100 COORD PTH ;
1652: L P[1652] 240cm/min CNT100 COORD PTH ;
1653: L P[1653] 240cm/min CNT100 COORD PTH ;
1654: L P[1654] 240cm/min CNT100 COORD PTH ;
1655: L P[1655] 240cm/min CNT100 COORD PTH ;
1656: L P[1656] 240cm/min CNT100 COORD PTH ;
1657: L P[1657] 240cm/min CNT100 COORD PTH ;
1658: L P[1658] 240cm/min CNT100 COORD PTH ;
1659: L P[1659] 240cm/min CNT100 COORD PTH ;
1660: L P[1660] 240cm/min CNT100 COORD PTH ;
1661: L P[1661] 240cm/min CNT100 COORD PTH ;
1662: L P[1662] 240cm/min CNT100 COORD PTH ;
1663: L P[1663] 240cm/min CNT100 COORD PTH ;
1664: L P[1664] 240cm/min CNT100 COORD PTH ;
1665: L P[1665] 240cm/min CNT100 COORD PTH ;
1666: L P[1666] 240cm/min CNT100 COORD PTH ;
1667: L P[1667] 240cm/min CNT100 COORD PTH ;
1668: L P[1668] 240cm/min CNT100 COORD PTH ;
1669: L P[1669] 240cm/min CNT100 COORD PTH ;
1670: L P[1670] 240cm/min CNT100 COORD PTH ;
1671: L P[1671] 240cm/min CNT100 COORD PTH ;
1672: L P[1672] 240cm/min CNT100 COORD PTH ;
1673: L P[1673] 240cm/min CNT100 COORD PTH ;
1674: L P[1674] 240cm/min CNT100 COORD PTH ;
1675: L P[1675] 240cm/min CNT100 COORD PTH ;
1676: L P[1676] 240cm/min CNT100 COORD PTH ;
1677: L P[1677] 240cm/min CNT100 COORD PTH ;
: Arc End[1];
1678: L P[1678] 240cm/min CNT100 COORD ;
: Arc Start[1];
1679: L P[1679] 240cm/min CNT100 COORD PTH ;
1680: L P[1680] 240cm/min CNT100 COORD PTH ;
1681: L P[1681] 240cm/min CNT100 COORD PTH ;
1682: L P[1682] 240cm/min CNT100 COORD PTH ;
1683: L P[1683] 240cm/min CNT100 COORD PTH ;
1684: L P[1684] 240cm/min CNT100 COORD PTH ;
1685: L P[1685] 240cm/min CNT100 COORD PTH ;
1686: L P[1686] 240cm/min CNT100 COORD PTH ;
1687: L P[1687] 240cm/min CNT100 COORD PTH ;
1688: L P[1688] 240cm/min CNT100 COORD PTH ;
1689: L P[1689] 240cm/min CNT100 COORD PTH ;
1690: L P[1690] 240cm/min CNT100 COORD PTH ;
1691: L P[1691] 240cm/min CNT100 COORD PTH ;
1692: L P[1692] 240cm/min CNT100 COORD PTH ;
1693: L P[1693] 240cm/min CNT100 COORD PTH ;
1694: L P[1694] 240cm/min CNT100 COORD PTH ;
1695: L P[1695] 240cm/min CNT100 COORD PTH ;
1696: L P[1696] 240cm/min CNT100 COORD PTH ;
1697: L P[1697] 240cm/min CNT100 COORD PTH ;
1698: L P[1698] 240cm/min CNT100 COORD PTH ;
1699: L P[1699] 240cm/min CNT100 COORD PTH ;
1700: L P[1700] 240cm/min CNT100 COORD PTH ;
1701: L P[1701] 240cm/min CNT100 COORD PTH ;
1702: L P[1702] 240cm/min CNT100 COORD PTH ;
1703: L P[1703] 240cm/min CNT100 COORD PTH ;
1704: L P[1704] 240cm/min CNT100 COORD PTH ;
1705: L P[1705] 240cm/min CNT100 COORD PTH ;
1706: L P[1706] 240cm/min CNT100 COORD PTH ;
1707: L P[1707] 240cm/min CNT100 COORD PTH ;
1708: L P[1708] 240cm/min CNT100 COORD PTH ;
1709: L P[1709] 240cm/min CNT100 COORD PTH ;
1710: L P[1710] 240cm/min CNT100 COORD PTH ;
1711: L P[1711] 240cm/min CNT100 COORD PTH ;
1712: L P[1712] 240cm/min CNT100 COORD PTH ;
1713: L P[1713] 240cm/min CNT100 COORD PTH ;
1714: L P[1714] 240cm/min CNT100 COORD PTH ;
1715: L P[1715] 240cm/min CNT100 COORD PTH ;
1716: L P[1716] 240cm/min CNT100 COORD PTH ;
1717: L P[1717] 240cm/min CNT100 COORD PTH ;
1718: L P[1718] 240cm/min CNT100 COORD PTH ;
1719: L P[1719] 240cm/min CNT100 COORD PTH ;
1720: L P[1720] 240cm/min CNT100 COORD PTH ;
1721: L P[1721] 240cm/min CNT100 COORD PTH ;
1722: L P[1722] 240cm/min CNT100 COORD PTH ;
1723: L P[1723] 240cm/min CNT100 COORD PTH ;
1724: L P[1724] 240cm/min CNT100 COORD PTH ;
1725: L P[1725] 240cm/min CNT100 COORD PTH ;
1726: L P[1726] 240cm/min CNT100 COORD PTH ;
1727: L P[1727] 240cm/min CNT100 COORD PTH ;
1728: L P[1728] 240cm/min CNT100 COORD PTH ;
1729: L P[1729] 240cm/min CNT100 COORD PTH ;
1730: L P[1730] 240cm/min CNT100 COORD PTH ;
1731: L P[1731] 240cm/min CNT100 COORD PTH ;
1732: L P[1732] 240cm/min CNT100 COORD PTH ;
1733: L P[1733] 240cm/min CNT100 COORD PTH ;
1734: L P[1734] 240cm/min CNT100 COORD PTH ;
1735: L P[1735] 240cm/min CNT100 COORD PTH ;
1736: L P[1736] 240cm/min CNT100 COORD PTH ;
1737: L P[1737] 240cm/min CNT100 COORD PTH ;
1738: L P[1738] 240cm/min CNT100 COORD PTH ;
1739: L P[1739] 240cm/min CNT100 COORD PTH ;
1740: L P[1740] 240cm/min CNT100 COORD PTH ;
1741: L P[1741] 240cm/min CNT100 COORD PTH ;
1742: L P[1742] 240cm/min CNT100 COORD PTH ;
1743: L P[1743] 240cm/min CNT100 COORD PTH ;
1744: L P[1744] 240cm/min CNT100 COORD PTH ;
1745: L P[1745] 240cm/min CNT100 COORD PTH ;
1746: L P[1746] 240cm/min CNT100 COORD PTH ;
1747: L P[1747] 240cm/min CNT100 COORD PTH ;
1748: L P[1748] 240cm/min CNT100 COORD PTH ;
1749: L P[1749] 240cm/min CNT100 COORD PTH ;
1750: L P[1750] 240cm/min CNT100 COORD PTH ;
1751: L P[1751] 240cm/min CNT100 COORD PTH ;
1752: L P[1752] 240cm/min CNT100 COORD PTH ;
1753: L P[1753] 240cm/min CNT100 COORD PTH ;
1754: L P[1754] 240cm/min CNT100 COORD PTH ;
1755: L P[1755] 240cm/min CNT100 COORD PTH ;
1756: L P[1756] 240cm/min CNT100 COORD PTH ;
1757: L P[1757] 240cm/min CNT100 COORD PTH ;
1758: L P[1758] 240cm/min CNT100 COORD PTH ;
1759: L P[1759] 240cm/min CNT100 COORD PTH ;
1760: L P[1760] 240cm/min CNT100 COORD PTH ;
1761: L P[1761] 240cm/min CNT100 COORD PTH ;
1762: L P[1762] 240cm/min CNT100 COORD PTH ;
1763: L P[1763] 240cm/min CNT100 COORD PTH ;
1764: L P[1764] 240cm/min CNT100 COORD PTH ;
1765: L P[1765] 240cm/min CNT100 COORD PTH ;
1766: L P[1766] 240cm/min CNT100 COORD PTH ;
1767: L P[1767] 240cm/min CNT100 COORD PTH ;
1768: L P[1768] 240cm/min CNT100 COORD PTH ;
1769: L P[1769] 240cm/min CNT100 COORD PTH ;
1770: L P[1770] 240cm/min CNT100 COORD PTH ;
1771: L P[1771] 240cm/min CNT100 COORD PTH ;
1772: L P[1772] 240cm/min CNT100 COORD PTH ;
1773: L P[1773] 240cm/min CNT100 COORD PTH ;
1774: L P[1774] 240cm/min CNT100 COORD PTH ;
1775: L P[1775] 240cm/min CNT100 COORD PTH ;
1776: L P[1776] 240cm/min CNT100 COORD PTH ;
1777: L P[1777] 240cm/min CNT100 COORD PTH ;
1778: L P[1778] 240cm/min CNT100 COORD PTH ;
1779: L P[1779] 240cm/min CNT100 COORD PTH ;
1780: L P[1780] 240cm/min CNT100 COORD PTH ;
1781: L P[1781] 240cm/min CNT100 COORD PTH ;
1782: L P[1782] 240cm/min CNT100 COORD PTH ;
: Arc End[1];
:R[34]=1;
:SR[23]=$SCR_GRP[1].$MCH_POS_X;
:SR[24]=$SCR_GRP[1].$MCH_POS_Y;
1793: L P[1793] 800cm/min CNT100 COORD ;
:SR[23]=$SCR_GRP[1].$MCH_POS_X;
:SR[24]=$SCR_GRP[1].$MCH_POS_Y;
1794: L P[1794] 800cm/min CNT100 COORD PTH ;
:SR[23]=$SCR_GRP[1].$MCH_POS_X;
:SR[24]=$SCR_GRP[1].$MCH_POS_Y;
1795: L P[1795] 800cm/min CNT100 COORD PTH ;
:SR[23]=$SCR_GRP[1].$MCH_POS_X;
:SR[24]=$SCR_GRP[1].$MCH_POS_Y;
1796: L P[1796] 800cm/min CNT100 COORD PTH ;
:SR[23]=$SCR_GRP[1].$MCH_POS_X;
:SR[24]=$SCR_GRP[1].$MCH_POS_Y;
1797: L P[1797] 800cm/min CNT100 COORD PTH ;
:SR[23]=$SCR_GRP[1].$MCH_POS_X;
:SR[24]=$SCR_GRP[1].$MCH_POS_Y;
1798: L P[1798] 800cm/min CNT100 COORD PTH ;
:SR[23]=$SCR_GRP[1].$MCH_POS_X;
:SR[24]=$SCR_GRP[1].$MCH_POS_Y;
1799: L P[1799] 800cm/min CNT100 COORD PTH ;
:SR[23]=$SCR_GRP[1].$MCH_POS_X;
:SR[24]=$SCR_GRP[1].$MCH_POS_Y;
1800: L P[1800] 800cm/min CNT100 COORD PTH ;
:SR[23]=$SCR_GRP[1].$MCH_POS_X;
:SR[24]=$SCR_GRP[1].$MCH_POS_Y;
1801: L P[1801] 800cm/min CNT100 COORD PTH ;
:SR[23]=$SCR_GRP[1].$MCH_POS_X;
:SR[24]=$SCR_GRP[1].$MCH_POS_Y;
1802: L P[1802] 800cm/min CNT100 COORD PTH ;
:SR[23]=$SCR_GRP[1].$MCH_POS_X;
:SR[24]=$SCR_GRP[1].$MCH_POS_Y;
1803: L P[1803] 800cm/min CNT100 COORD PTH ;
:SR[23]=$SCR_GRP[1].$MCH_POS_X;
:SR[24]=$SCR_GRP[1].$MCH_POS_Y;
1804: L P[1804] 800cm/min CNT100 COORD PTH ;
:SR[23]=$SCR_GRP[1].$MCH_POS_X;
:SR[24]=$SCR_GRP[1].$MCH_POS_Y;
1805: L P[1805] 800cm/min CNT100 COORD PTH ;
:SR[23]=$SCR_GRP[1].$MCH_POS_X;
:SR[24]=$SCR_GRP[1].$MCH_POS_Y;
1806: L P[1806] 800cm/min CNT100 COORD PTH ;
:SR[23]=$SCR_GRP[1].$MCH_POS_X;
:SR[24]=$SCR_GRP[1].$MCH_POS_Y;
1807: L P[1807] 800cm/min CNT100 COORD PTH ;
:SR[23]=$SCR_GRP[1].$MCH_POS_X;
:SR[24]=$SCR_GRP[1].$MCH_POS_Y;
1808: L P[1808] 800cm/min CNT100 COORD PTH ;
:SR[23]=$SCR_GRP[1].$MCH_POS_X;
:SR[24]=$SCR_GRP[1].$MCH_POS_Y;
1809: L P[1809] 800cm/min CNT100 COORD PTH ;
:SR[23]=$SCR_GRP[1].$MCH_POS_X;
:SR[24]=$SCR_GRP[1].$MCH_POS_Y;
1810: L P[1810] 800cm/min CNT100 COORD PTH ;
:SR[23]=$SCR_GRP[1].$MCH_POS_X;
:SR[24]=$SCR_GRP[1].$MCH_POS_Y;
1811: L P[1811] 800cm/min CNT100 COORD PTH ;
:SR[23]=$SCR_GRP[1].$MCH_POS_X;
:SR[24]=$SCR_GRP[1].$MCH_POS_Y;
1812: L P[1812] 800cm/min CNT100 COORD PTH ;
:SR[23]=$SCR_GRP[1].$MCH_POS_X;
:SR[24]=$SCR_GRP[1].$MCH_POS_Y;
1813: L P[1813] 800cm/min CNT100 COORD PTH ;
:SR[23]=$SCR_GRP[1].$MCH_POS_X;
:SR[24]=$SCR_GRP[1].$MCH_POS_Y;
1814: L P[1814] 800cm/min CNT100 COORD PTH ;
:SR[23]=$SCR_GRP[1].$MCH_POS_X;
:SR[24]=$SCR_GRP[1].$MCH_POS_Y;
1815: L P[1815] 800cm/min CNT100 COORD PTH ;
:SR[23]=$SCR_GRP[1].$MCH_POS_X;
:SR[24]=$SCR_GRP[1].$MCH_POS_Y;
1816: L P[1816] 800cm/min CNT100 COORD PTH ;
:SR[23]=$SCR_GRP[1].$MCH_POS_X;
:SR[24]=$SCR_GRP[1].$MCH_POS_Y;
1817: L P[1817] 800cm/min CNT100 COORD PTH ;
:SR[23]=$SCR_GRP[1].$MCH_POS_X;
:SR[24]=$SCR_GRP[1].$MCH_POS_Y;
1818: L P[1818] 800cm/min CNT100 COORD PTH ;
:SR[23]=$SCR_GRP[1].$MCH_POS_X;
:SR[24]=$SCR_GRP[1].$MCH_POS_Y;
1819: L P[1819] 800cm/min CNT100 COORD PTH ;
:SR[23]=$SCR_GRP[1].$MCH_POS_X;
:SR[24]=$SCR_GRP[1].$MCH_POS_Y;
1820: L P[1820] 800cm/min CNT100 COORD PTH ;
:SR[23]=$SCR_GRP[1].$MCH_POS_X;
:SR[24]=$SCR_GRP[1].$MCH_POS_Y;
1821: L P[1821] 800cm/min CNT100 COORD PTH ;
:SR[23]=$SCR_GRP[1].$MCH_POS_X;
:SR[24]=$SCR_GRP[1].$MCH_POS_Y;
1822: L P[1822] 800cm/min CNT100 COORD PTH ;
:SR[23]=$SCR_GRP[1].$MCH_POS_X;
:SR[24]=$SCR_GRP[1].$MCH_POS_Y;
1823: L P[1823] 800cm/min CNT100 COORD PTH ;
:SR[23]=$SCR_GRP[1].$MCH_POS_X;
:SR[24]=$SCR_GRP[1].$MCH_POS_Y;
1824: L P[1824] 800cm/min CNT100 COORD PTH ;
:SR[23]=$SCR_GRP[1].$MCH_POS_X;
:SR[24]=$SCR_GRP[1].$MCH_POS_Y;
1825: L P[1825] 800cm/min CNT100 COORD PTH ;
:SR[23]=$SCR_GRP[1].$MCH_POS_X;
:SR[24]=$SCR_GRP[1].$MCH_POS_Y;
1826: L P[1826] 800cm/min CNT100 COORD PTH ;
:SR[23]=$SCR_GRP[1].$MCH_POS_X;
:SR[24]=$SCR_GRP[1].$MCH_POS_Y;
1827: L P[1827] 800cm/min CNT100 COORD PTH ;
:SR[23]=$SCR_GRP[1].$MCH_POS_X;
:SR[24]=$SCR_GRP[1].$MCH_POS_Y;
1828: L P[1828] 800cm/min CNT100 COORD PTH ;
:SR[23]=$SCR_GRP[1].$MCH_POS_X;
:SR[24]=$SCR_GRP[1].$MCH_POS_Y;
1829: L P[1829] 800cm/min CNT100 COORD PTH ;
:SR[23]=$SCR_GRP[1].$MCH_POS_X;
:SR[24]=$SCR_GRP[1].$MCH_POS_Y;
1830: L P[1830] 800cm/min CNT100 COORD PTH ;
:SR[23]=$SCR_GRP[1].$MCH_POS_X;
:SR[24]=$SCR_GRP[1].$MCH_POS_Y;
1831: L P[1831] 800cm/min CNT100 COORD PTH ;
:SR[23]=$SCR_GRP[1].$MCH_POS_X;
:SR[24]=$SCR_GRP[1].$MCH_POS_Y;
1832: L P[1832] 800cm/min CNT100 COORD PTH ;
:SR[23]=$SCR_GRP[1].$MCH_POS_X;
:SR[24]=$SCR_GRP[1].$MCH_POS_Y;
1833: L P[1833] 800cm/min CNT100 COORD PTH ;
:SR[23]=$SCR_GRP[1].$MCH_POS_X;
:SR[24]=$SCR_GRP[1].$MCH_POS_Y;
1834: L P[1834] 800cm/min CNT100 COORD PTH ;
:SR[23]=$SCR_GRP[1].$MCH_POS_X;
:SR[24]=$SCR_GRP[1].$MCH_POS_Y;
1835: L P[1835] 800cm/min CNT100 COORD PTH ;
:SR[23]=$SCR_GRP[1].$MCH_POS_X;
:SR[24]=$SCR_GRP[1].$MCH_POS_Y;
1836: L P[1836] 800cm/min CNT100 COORD PTH ;
:SR[23]=$SCR_GRP[1].$MCH_POS_X;
:SR[24]=$SCR_GRP[1].$MCH_POS_Y;
1837: L P[1837] 800cm/min CNT100 COORD PTH ;
:SR[23]=$SCR_GRP[1].$MCH_POS_X;
:SR[24]=$SCR_GRP[1].$MCH_POS_Y;
1838: L P[1838] 800cm/min CNT100 COORD PTH ;
:SR[23]=$SCR_GRP[1].$MCH_POS_X;
:SR[24]=$SCR_GRP[1].$MCH_POS_Y;
1839: L P[1839] 800cm/min CNT100 COORD PTH ;
:SR[23]=$SCR_GRP[1].$MCH_POS_X;
:SR[24]=$SCR_GRP[1].$MCH_POS_Y;
1840: L P[1840] 800cm/min CNT100 COORD PTH ;
:SR[23]=$SCR_GRP[1].$MCH_POS_X;
:SR[24]=$SCR_GRP[1].$MCH_POS_Y;
1841: L P[1841] 800cm/min CNT100 COORD PTH ;
:SR[23]=$SCR_GRP[1].$MCH_POS_X;
:SR[24]=$SCR_GRP[1].$MCH_POS_Y;
1842: L P[1842] 800cm/min CNT100 COORD PTH ;
:SR[23]=$SCR_GRP[1].$MCH_POS_X;
:SR[24]=$SCR_GRP[1].$MCH_POS_Y;
1843: L P[1843] 800cm/min CNT100 COORD PTH ;
:SR[23]=$SCR_GRP[1].$MCH_POS_X;
:SR[24]=$SCR_GRP[1].$MCH_POS_Y;
1844: L P[1844] 800cm/min CNT100 COORD PTH ;
:SR[23]=$SCR_GRP[1].$MCH_POS_X;
:SR[24]=$SCR_GRP[1].$MCH_POS_Y;
1845: L P[1845] 800cm/min CNT100 COORD PTH ;
:SR[23]=$SCR_GRP[1].$MCH_POS_X;
:SR[24]=$SCR_GRP[1].$MCH_POS_Y;
1846: L P[1846] 800cm/min CNT100 COORD PTH ;
:SR[23]=$SCR_GRP[1].$MCH_POS_X;
:SR[24]=$SCR_GRP[1].$MCH_POS_Y;
1847: L P[1847] 800cm/min CNT100 COORD PTH ;
:SR[23]=$SCR_GRP[1].$MCH_POS_X;
:SR[24]=$SCR_GRP[1].$MCH_POS_Y;
1848: L P[1848] 800cm/min CNT100 COORD PTH ;
:SR[23]=$SCR_GRP[1].$MCH_POS_X;
:SR[24]=$SCR_GRP[1].$MCH_POS_Y;
1849: L P[1849] 800cm/min CNT100 COORD PTH ;
:SR[23]=$SCR_GRP[1].$MCH_POS_X;
:SR[24]=$SCR_GRP[1].$MCH_POS_Y;
1850: L P[1850] 800cm/min CNT100 COORD PTH ;
:SR[23]=$SCR_GRP[1].$MCH_POS_X;
:SR[24]=$SCR_GRP[1].$MCH_POS_Y;
1851: L P[1851] 800cm/min CNT100 COORD PTH ;
:SR[23]=$SCR_GRP[1].$MCH_POS_X;
:SR[24]=$SCR_GRP[1].$MCH_POS_Y;
1852: L P[1852] 800cm/min CNT100 COORD PTH ;
:SR[23]=$SCR_GRP[1].$MCH_POS_X;
:SR[24]=$SCR_GRP[1].$MCH_POS_Y;
1853: L P[1853] 800cm/min CNT100 COORD PTH ;
:SR[23]=$SCR_GRP[1].$MCH_POS_X;
:SR[24]=$SCR_GRP[1].$MCH_POS_Y;
1854: L P[1854] 800cm/min CNT100 COORD PTH ;
:SR[23]=$SCR_GRP[1].$MCH_POS_X;
:SR[24]=$SCR_GRP[1].$MCH_POS_Y;
1855: L P[1855] 800cm/min CNT100 COORD PTH ;
:SR[23]=$SCR_GRP[1].$MCH_POS_X;
:SR[24]=$SCR_GRP[1].$MCH_POS_Y;
1856: L P[1856] 800cm/min CNT100 COORD PTH ;
:SR[23]=$SCR_GRP[1].$MCH_POS_X;
:SR[24]=$SCR_GRP[1].$MCH_POS_Y;
1857: L P[1857] 800cm/min CNT100 COORD PTH ;
:SR[23]=$SCR_GRP[1].$MCH_POS_X;
:SR[24]=$SCR_GRP[1].$MCH_POS_Y;
1858: L P[1858] 800cm/min CNT100 COORD PTH ;
:SR[23]=$SCR_GRP[1].$MCH_POS_X;
:SR[24]=$SCR_GRP[1].$MCH_POS_Y;
1859: L P[1859] 800cm/min CNT100 COORD PTH ;
:SR[23]=$SCR_GRP[1].$MCH_POS_X;
:SR[24]=$SCR_GRP[1].$MCH_POS_Y;
1860: L P[1860] 800cm/min CNT100 COORD PTH ;
:SR[23]=$SCR_GRP[1].$MCH_POS_X;
:SR[24]=$SCR_GRP[1].$MCH_POS_Y;
1861: L P[1861] 800cm/min CNT100 COORD PTH ;
:SR[23]=$SCR_GRP[1].$MCH_POS_X;
:SR[24]=$SCR_GRP[1].$MCH_POS_Y;
1862: L P[1862] 800cm/min CNT100 COORD PTH ;
:SR[23]=$SCR_GRP[1].$MCH_POS_X;
:SR[24]=$SCR_GRP[1].$MCH_POS_Y;
1863: L P[1863] 800cm/min CNT100 COORD PTH ;
:SR[23]=$SCR_GRP[1].$MCH_POS_X;
:SR[24]=$SCR_GRP[1].$MCH_POS_Y;
1864: L P[1864] 800cm/min CNT100 COORD PTH ;
:SR[23]=$SCR_GRP[1].$MCH_POS_X;
:SR[24]=$SCR_GRP[1].$MCH_POS_Y;
1865: L P[1865] 800cm/min CNT100 COORD PTH ;
:SR[23]=$SCR_GRP[1].$MCH_POS_X;
:SR[24]=$SCR_GRP[1].$MCH_POS_Y;
1866: L P[1866] 800cm/min CNT100 COORD PTH ;
:SR[23]=$SCR_GRP[1].$MCH_POS_X;
:SR[24]=$SCR_GRP[1].$MCH_POS_Y;
1867: L P[1867] 800cm/min CNT100 COORD PTH ;
:SR[23]=$SCR_GRP[1].$MCH_POS_X;
:SR[24]=$SCR_GRP[1].$MCH_POS_Y;
1868: L P[1868] 800cm/min CNT100 COORD PTH ;
:SR[23]=$SCR_GRP[1].$MCH_POS_X;
:SR[24]=$SCR_GRP[1].$MCH_POS_Y;
1869: L P[1869] 800cm/min CNT100 COORD PTH ;
:SR[23]=$SCR_GRP[1].$MCH_POS_X;
:SR[24]=$SCR_GRP[1].$MCH_POS_Y;
1870: L P[1870] 800cm/min CNT100 COORD PTH ;
:SR[23]=$SCR_GRP[1].$MCH_POS_X;
:SR[24]=$SCR_GRP[1].$MCH_POS_Y;
1871: L P[1871] 800cm/min CNT100 COORD PTH ;
:SR[23]=$SCR_GRP[1].$MCH_POS_X;
:SR[24]=$SCR_GRP[1].$MCH_POS_Y;
1872: L P[1872] 800cm/min CNT100 COORD PTH ;
:SR[23]=$SCR_GRP[1].$MCH_POS_X;
:SR[24]=$SCR_GRP[1].$MCH_POS_Y;
1873: L P[1873] 800cm/min CNT100 COORD PTH ;
:SR[23]=$SCR_GRP[1].$MCH_POS_X;
:SR[24]=$SCR_GRP[1].$MCH_POS_Y;
1874: L P[1874] 800cm/min CNT100 COORD PTH ;
:SR[23]=$SCR_GRP[1].$MCH_POS_X;
:SR[24]=$SCR_GRP[1].$MCH_POS_Y;
1875: L P[1875] 800cm/min CNT100 COORD PTH ;
:SR[23]=$SCR_GRP[1].$MCH_POS_X;
:SR[24]=$SCR_GRP[1].$MCH_POS_Y;
1876: L P[1876] 800cm/min CNT100 COORD PTH ;
:SR[23]=$SCR_GRP[1].$MCH_POS_X;
:SR[24]=$SCR_GRP[1].$MCH_POS_Y;
1877: L P[1877] 800cm/min CNT100 COORD PTH ;
:SR[23]=$SCR_GRP[1].$MCH_POS_X;
:SR[24]=$SCR_GRP[1].$MCH_POS_Y;
1878: L P[1878] 800cm/min CNT100 COORD PTH ;
:SR[23]=$SCR_GRP[1].$MCH_POS_X;
:SR[24]=$SCR_GRP[1].$MCH_POS_Y;
1879: L P[1879] 800cm/min CNT100 COORD PTH ;
:SR[23]=$SCR_GRP[1].$MCH_POS_X;
:SR[24]=$SCR_GRP[1].$MCH_POS_Y;
1880: L P[1880] 800cm/min CNT100 COORD PTH ;
:SR[23]=$SCR_GRP[1].$MCH_POS_X;
:SR[24]=$SCR_GRP[1].$MCH_POS_Y;
1881: L P[1881] 800cm/min CNT100 COORD PTH ;
:SR[23]=$SCR_GRP[1].$MCH_POS_X;
:SR[24]=$SCR_GRP[1].$MCH_POS_Y;
1882: L P[1882] 800cm/min CNT100 COORD PTH ;
:SR[23]=$SCR_GRP[1].$MCH_POS_X;
:SR[24]=$SCR_GRP[1].$MCH_POS_Y;
1883: L P[1883] 800cm/min CNT100 COORD PTH ;
:SR[23]=$SCR_GRP[1].$MCH_POS_X;
:SR[24]=$SCR_GRP[1].$MCH_POS_Y;
1884: L P[1884] 800cm/min CNT100 COORD PTH ;
:SR[23]=$SCR_GRP[1].$MCH_POS_X;
:SR[24]=$SCR_GRP[1].$MCH_POS_Y;
1885: L P[1885] 800cm/min CNT100 COORD PTH ;
:SR[23]=$SCR_GRP[1].$MCH_POS_X;
:SR[24]=$SCR_GRP[1].$MCH_POS_Y;
1886: L P[1886] 800cm/min CNT100 COORD PTH ;
:SR[23]=$SCR_GRP[1].$MCH_POS_X;
:SR[24]=$SCR_GRP[1].$MCH_POS_Y;
1887: L P[1887] 800cm/min CNT100 COORD PTH ;
:SR[23]=$SCR_GRP[1].$MCH_POS_X;
:SR[24]=$SCR_GRP[1].$MCH_POS_Y;
1888: L P[1888] 800cm/min CNT100 COORD PTH ;
:SR[23]=$SCR_GRP[1].$MCH_POS_X;
:SR[24]=$SCR_GRP[1].$MCH_POS_Y;
1889: L P[1889] 800cm/min CNT100 COORD PTH ;
:SR[23]=$SCR_GRP[1].$MCH_POS_X;
:SR[24]=$SCR_GRP[1].$MCH_POS_Y;
1890: L P[1890] 800cm/min CNT100 COORD PTH ;
:SR[23]=$SCR_GRP[1].$MCH_POS_X;
:SR[24]=$SCR_GRP[1].$MCH_POS_Y;
1891: L P[1891] 800cm/min CNT100 COORD PTH ;
:SR[23]=$SCR_GRP[1].$MCH_POS_X;
:SR[24]=$SCR_GRP[1].$MCH_POS_Y;
1892: L P[1892] 800cm/min CNT100 COORD PTH ;
:SR[23]=$SCR_GRP[1].$MCH_POS_X;
:SR[24]=$SCR_GRP[1].$MCH_POS_Y;
1893: L P[1893] 800cm/min CNT100 COORD PTH ;
:SR[23]=$SCR_GRP[1].$MCH_POS_X;
:SR[24]=$SCR_GRP[1].$MCH_POS_Y;
1894: L P[1894] 800cm/min CNT100 COORD PTH ;
:SR[23]=$SCR_GRP[1].$MCH_POS_X;
:SR[24]=$SCR_GRP[1].$MCH_POS_Y;
1895: L P[1895] 800cm/min CNT100 COORD PTH ;
:SR[23]=$SCR_GRP[1].$MCH_POS_X;
:SR[24]=$SCR_GRP[1].$MCH_POS_Y;
1896: L P[1896] 800cm/min CNT100 COORD PTH ;
:SR[23]=$SCR_GRP[1].$MCH_POS_X;
:SR[24]=$SCR_GRP[1].$MCH_POS_Y;
1897: L P[1897] 800cm/min CNT100 COORD PTH ;
:SR[23]=$SCR_GRP[1].$MCH_POS_X;
:SR[24]=$SCR_GRP[1].$MCH_POS_Y;
1898: L P[1898] 800cm/min CNT100 COORD PTH ;
:SR[23]=$SCR_GRP[1].$MCH_POS_X;
:SR[24]=$SCR_GRP[1].$MCH_POS_Y;
1899: L P[1899] 800cm/min CNT100 COORD PTH ;
:SR[23]=$SCR_GRP[1].$MCH_POS_X;
:SR[24]=$SCR_GRP[1].$MCH_POS_Y;
1900: L P[1900] 800cm/min CNT100 COORD PTH ;
:SR[23]=$SCR_GRP[1].$MCH_POS_X;
:SR[24]=$SCR_GRP[1].$MCH_POS_Y;
1901: L P[1901] 800cm/min CNT100 COORD PTH ;
:SR[23]=$SCR_GRP[1].$MCH_POS_X;
:SR[24]=$SCR_GRP[1].$MCH_POS_Y;
1902: L P[1902] 800cm/min CNT100 COORD PTH ;
:SR[23]=$SCR_GRP[1].$MCH_POS_X;
:SR[24]=$SCR_GRP[1].$MCH_POS_Y;
1903: L P[1903] 800cm/min CNT100 COORD PTH ;
:SR[23]=$SCR_GRP[1].$MCH_POS_X;
:SR[24]=$SCR_GRP[1].$MCH_POS_Y;
1904: L P[1904] 800cm/min CNT100 COORD PTH ;
:SR[23]=$SCR_GRP[1].$MCH_POS_X;
:SR[24]=$SCR_GRP[1].$MCH_POS_Y;
1905: L P[1905] 800cm/min CNT100 COORD PTH ;
:SR[23]=$SCR_GRP[1].$MCH_POS_X;
:SR[24]=$SCR_GRP[1].$MCH_POS_Y;
1906: L P[1906] 800cm/min CNT100 COORD PTH ;
:SR[23]=$SCR_GRP[1].$MCH_POS_X;
:SR[24]=$SCR_GRP[1].$MCH_POS_Y;
1907: L P[1907] 800cm/min CNT100 COORD PTH ;
:SR[23]=$SCR_GRP[1].$MCH_POS_X;
:SR[24]=$SCR_GRP[1].$MCH_POS_Y;
1908: L P[1908] 800cm/min CNT100 COORD PTH ;
:SR[23]=$SCR_GRP[1].$MCH_POS_X;
:SR[24]=$SCR_GRP[1].$MCH_POS_Y;
1909: L P[1909] 800cm/min CNT100 COORD PTH ;
:SR[23]=$SCR_GRP[1].$MCH_POS_X;
:SR[24]=$SCR_GRP[1].$MCH_POS_Y;
1910: L P[1910] 800cm/min CNT100 COORD PTH ;
:SR[23]=$SCR_GRP[1].$MCH_POS_X;
:SR[24]=$SCR_GRP[1].$MCH_POS_Y;
1911: L P[1911] 800cm/min CNT100 COORD PTH ;
:SR[23]=$SCR_GRP[1].$MCH_POS_X;
:SR[24]=$SCR_GRP[1].$MCH_POS_Y;
1912: L P[1912] 800cm/min CNT100 COORD PTH ;
:SR[23]=$SCR_GRP[1].$MCH_POS_X;
:SR[24]=$SCR_GRP[1].$MCH_POS_Y;
1913: L P[1913] 800cm/min CNT100 COORD PTH ;
:SR[23]=$SCR_GRP[1].$MCH_POS_X;
:SR[24]=$SCR_GRP[1].$MCH_POS_Y;
1914: L P[1914] 800cm/min CNT100 COORD PTH ;
:SR[23]=$SCR_GRP[1].$MCH_POS_X;
:SR[24]=$SCR_GRP[1].$MCH_POS_Y;
1915: L P[1915] 800cm/min CNT100 COORD PTH ;
:SR[23]=$SCR_GRP[1].$MCH_POS_X;
:SR[24]=$SCR_GRP[1].$MCH_POS_Y;
1916: L P[1916] 800cm/min CNT100 COORD PTH ;
:SR[23]=$SCR_GRP[1].$MCH_POS_X;
:SR[24]=$SCR_GRP[1].$MCH_POS_Y;
1917: L P[1917] 800cm/min CNT100 COORD PTH ;
:SR[23]=$SCR_GRP[1].$MCH_POS_X;
:SR[24]=$SCR_GRP[1].$MCH_POS_Y;
1918: L P[1918] 800cm/min CNT100 COORD PTH ;
:SR[23]=$SCR_GRP[1].$MCH_POS_X;
:SR[24]=$SCR_GRP[1].$MCH_POS_Y;
1919: L P[1919] 800cm/min CNT100 COORD PTH ;
:SR[23]=$SCR_GRP[1].$MCH_POS_X;
:SR[24]=$SCR_GRP[1].$MCH_POS_Y;
1920: L P[1920] 800cm/min CNT100 COORD PTH ;
:SR[23]=$SCR_GRP[1].$MCH_POS_X;
:SR[24]=$SCR_GRP[1].$MCH_POS_Y;
1921: L P[1921] 800cm/min CNT100 COORD PTH ;
:SR[23]=$SCR_GRP[1].$MCH_POS_X;
:SR[24]=$SCR_GRP[1].$MCH_POS_Y;
1922: L P[1922] 800cm/min CNT100 COORD PTH ;
:SR[23]=$SCR_GRP[1].$MCH_POS_X;
:SR[24]=$SCR_GRP[1].$MCH_POS_Y;
1923: L P[1923] 800cm/min CNT100 COORD PTH ;
:SR[23]=$SCR_GRP[1].$MCH_POS_X;
:SR[24]=$SCR_GRP[1].$MCH_POS_Y;
1924: L P[1924] 800cm/min CNT100 COORD PTH ;
:SR[23]=$SCR_GRP[1].$MCH_POS_X;
:SR[24]=$SCR_GRP[1].$MCH_POS_Y;
1925: L P[1925] 800cm/min CNT100 COORD PTH ;
:SR[23]=$SCR_GRP[1].$MCH_POS_X;
:SR[24]=$SCR_GRP[1].$MCH_POS_Y;
1926: L P[1926] 800cm/min CNT100 COORD PTH ;
:SR[23]=$SCR_GRP[1].$MCH_POS_X;
:SR[24]=$SCR_GRP[1].$MCH_POS_Y;
1927: L P[1927] 800cm/min CNT100 COORD PTH ;
:SR[23]=$SCR_GRP[1].$MCH_POS_X;
:SR[24]=$SCR_GRP[1].$MCH_POS_Y;
1928: L P[1928] 800cm/min CNT100 COORD PTH ;
:SR[23]=$SCR_GRP[1].$MCH_POS_X;
:SR[24]=$SCR_GRP[1].$MCH_POS_Y;
1929: L P[1929] 800cm/min CNT100 COORD PTH ;
:SR[23]=$SCR_GRP[1].$MCH_POS_X;
:SR[24]=$SCR_GRP[1].$MCH_POS_Y;
1930: L P[1930] 800cm/min CNT100 COORD PTH ;
:SR[23]=$SCR_GRP[1].$MCH_POS_X;
:SR[24]=$SCR_GRP[1].$MCH_POS_Y;
1931: L P[1931] 800cm/min CNT100 COORD PTH ;
:SR[23]=$SCR_GRP[1].$MCH_POS_X;
:SR[24]=$SCR_GRP[1].$MCH_POS_Y;
1932: L P[1932] 800cm/min CNT100 COORD PTH ;
:SR[23]=$SCR_GRP[1].$MCH_POS_X;
:SR[24]=$SCR_GRP[1].$MCH_POS_Y;
1933: L P[1933] 800cm/min CNT100 COORD PTH ;
:SR[23]=$SCR_GRP[1].$MCH_POS_X;
:SR[24]=$SCR_GRP[1].$MCH_POS_Y;
1934: L P[1934] 800cm/min CNT100 COORD PTH ;
:SR[23]=$SCR_GRP[1].$MCH_POS_X;
:SR[24]=$SCR_GRP[1].$MCH_POS_Y;
1935: L P[1935] 800cm/min CNT100 COORD PTH ;
:SR[23]=$SCR_GRP[1].$MCH_POS_X;
:SR[24]=$SCR_GRP[1].$MCH_POS_Y;
1936: L P[1936] 800cm/min CNT100 COORD PTH ;
:SR[23]=$SCR_GRP[1].$MCH_POS_X;
:SR[24]=$SCR_GRP[1].$MCH_POS_Y;
1937: L P[1937] 800cm/min CNT100 COORD PTH ;
:SR[23]=$SCR_GRP[1].$MCH_POS_X;
:SR[24]=$SCR_GRP[1].$MCH_POS_Y;
1938: L P[1938] 800cm/min CNT100 COORD PTH ;
:SR[23]=$SCR_GRP[1].$MCH_POS_X;
:SR[24]=$SCR_GRP[1].$MCH_POS_Y;
1939: L P[1939] 800cm/min CNT100 COORD PTH ;
:SR[23]=$SCR_GRP[1].$MCH_POS_X;
:SR[24]=$SCR_GRP[1].$MCH_POS_Y;
1940: L P[1940] 800cm/min CNT100 COORD PTH ;
:SR[23]=$SCR_GRP[1].$MCH_POS_X;
:SR[24]=$SCR_GRP[1].$MCH_POS_Y;
1941: L P[1941] 800cm/min CNT100 COORD PTH ;
:SR[23]=$SCR_GRP[1].$MCH_POS_X;
:SR[24]=$SCR_GRP[1].$MCH_POS_Y;
1942: L P[1942] 800cm/min CNT100 COORD PTH ;
:SR[23]=$SCR_GRP[1].$MCH_POS_X;
:SR[24]=$SCR_GRP[1].$MCH_POS_Y;
1943: L P[1943] 800cm/min CNT100 COORD PTH ;
:SR[23]=$SCR_GRP[1].$MCH_POS_X;
:SR[24]=$SCR_GRP[1].$MCH_POS_Y;
1944: L P[1944] 800cm/min CNT100 COORD PTH ;
:SR[23]=$SCR_GRP[1].$MCH_POS_X;
:SR[24]=$SCR_GRP[1].$MCH_POS_Y;
1945: L P[1945] 800cm/min CNT100 COORD PTH ;
:SR[23]=$SCR_GRP[1].$MCH_POS_X;
:SR[24]=$SCR_GRP[1].$MCH_POS_Y;
1946: L P[1946] 800cm/min CNT100 COORD PTH ;
:SR[23]=$SCR_GRP[1].$MCH_POS_X;
:SR[24]=$SCR_GRP[1].$MCH_POS_Y;
1947: L P[1947] 800cm/min CNT100 COORD PTH ;
:SR[23]=$SCR_GRP[1].$MCH_POS_X;
:SR[24]=$SCR_GRP[1].$MCH_POS_Y;
1948: L P[1948] 800cm/min CNT100 COORD PTH ;
:SR[23]=$SCR_GRP[1].$MCH_POS_X;
:SR[24]=$SCR_GRP[1].$MCH_POS_Y;
1949: L P[1949] 800cm/min CNT100 COORD PTH ;
:SR[23]=$SCR_GRP[1].$MCH_POS_X;
:SR[24]=$SCR_GRP[1].$MCH_POS_Y;
1950: L P[1950] 800cm/min CNT100 COORD PTH ;
:SR[23]=$SCR_GRP[1].$MCH_POS_X;
:SR[24]=$SCR_GRP[1].$MCH_POS_Y;
1951: L P[1951] 800cm/min CNT100 COORD PTH ;
:SR[23]=$SCR_GRP[1].$MCH_POS_X;
:SR[24]=$SCR_GRP[1].$MCH_POS_Y;
1952: L P[1952] 800cm/min CNT100 COORD PTH ;
:SR[23]=$SCR_GRP[1].$MCH_POS_X;
:SR[24]=$SCR_GRP[1].$MCH_POS_Y;
1953: L P[1953] 800cm/min CNT100 COORD PTH ;
:SR[23]=$SCR_GRP[1].$MCH_POS_X;
:SR[24]=$SCR_GRP[1].$MCH_POS_Y;
1954: L P[1954] 800cm/min CNT100 COORD PTH ;
:SR[23]=$SCR_GRP[1].$MCH_POS_X;
:SR[24]=$SCR_GRP[1].$MCH_POS_Y;
1955: L P[1955] 800cm/min CNT100 COORD PTH ;
:SR[23]=$SCR_GRP[1].$MCH_POS_X;
:SR[24]=$SCR_GRP[1].$MCH_POS_Y;
1956: L P[1956] 800cm/min CNT100 COORD PTH ;
:SR[23]=$SCR_GRP[1].$MCH_POS_X;
:SR[24]=$SCR_GRP[1].$MCH_POS_Y;
1957: L P[1957] 800cm/min CNT100 COORD PTH ;
:SR[23]=$SCR_GRP[1].$MCH_POS_X;
:SR[24]=$SCR_GRP[1].$MCH_POS_Y;
1958: L P[1958] 800cm/min CNT100 COORD PTH ;
:SR[23]=$SCR_GRP[1].$MCH_POS_X;
:SR[24]=$SCR_GRP[1].$MCH_POS_Y;
1959: L P[1959] 800cm/min CNT100 COORD PTH ;
:SR[23]=$SCR_GRP[1].$MCH_POS_X;
:SR[24]=$SCR_GRP[1].$MCH_POS_Y;
1960: L P[1960] 800cm/min CNT100 COORD PTH ;
:SR[23]=$SCR_GRP[1].$MCH_POS_X;
:SR[24]=$SCR_GRP[1].$MCH_POS_Y;
1961: L P[1961] 800cm/min CNT100 COORD PTH ;
:SR[23]=$SCR_GRP[1].$MCH_POS_X;
:SR[24]=$SCR_GRP[1].$MCH_POS_Y;
1962: L P[1962] 800cm/min CNT100 COORD PTH ;
:SR[23]=$SCR_GRP[1].$MCH_POS_X;
:SR[24]=$SCR_GRP[1].$MCH_POS_Y;
1963: L P[1963] 800cm/min CNT100 COORD PTH ;
:SR[23]=$SCR_GRP[1].$MCH_POS_X;
:SR[24]=$SCR_GRP[1].$MCH_POS_Y;
1964: L P[1964] 800cm/min CNT100 COORD PTH ;
:SR[23]=$SCR_GRP[1].$MCH_POS_X;
:SR[24]=$SCR_GRP[1].$MCH_POS_Y;
1965: L P[1965] 800cm/min CNT100 COORD PTH ;
:SR[23]=$SCR_GRP[1].$MCH_POS_X;
:SR[24]=$SCR_GRP[1].$MCH_POS_Y;
1966: L P[1966] 800cm/min CNT100 COORD PTH ;
:SR[23]=$SCR_GRP[1].$MCH_POS_X;
:SR[24]=$SCR_GRP[1].$MCH_POS_Y;
1967: L P[1967] 800cm/min CNT100 COORD PTH ;
:SR[23]=$SCR_GRP[1].$MCH_POS_X;
:SR[24]=$SCR_GRP[1].$MCH_POS_Y;
1968: L P[1968] 800cm/min CNT100 COORD PTH ;
:SR[23]=$SCR_GRP[1].$MCH_POS_X;
:SR[24]=$SCR_GRP[1].$MCH_POS_Y;
1969: L P[1969] 800cm/min CNT100 COORD PTH ;
:SR[23]=$SCR_GRP[1].$MCH_POS_X;
:SR[24]=$SCR_GRP[1].$MCH_POS_Y;
1970: L P[1970] 800cm/min CNT100 COORD PTH ;
:SR[23]=$SCR_GRP[1].$MCH_POS_X;
:SR[24]=$SCR_GRP[1].$MCH_POS_Y;
1971: L P[1971] 800cm/min CNT100 COORD PTH ;
:SR[23]=$SCR_GRP[1].$MCH_POS_X;
:SR[24]=$SCR_GRP[1].$MCH_POS_Y;
1972: L P[1972] 800cm/min CNT100 COORD PTH ;
:SR[23]=$SCR_GRP[1].$MCH_POS_X;
:SR[24]=$SCR_GRP[1].$MCH_POS_Y;
1973: L P[1973] 800cm/min CNT100 COORD PTH ;
:SR[23]=$SCR_GRP[1].$MCH_POS_X;
:SR[24]=$SCR_GRP[1].$MCH_POS_Y;
1974: L P[1974] 800cm/min CNT100 COORD PTH ;
:SR[23]=$SCR_GRP[1].$MCH_POS_X;
:SR[24]=$SCR_GRP[1].$MCH_POS_Y;
1975: L P[1975] 800cm/min CNT100 COORD PTH ;
:SR[23]=$SCR_GRP[1].$MCH_POS_X;
:SR[24]=$SCR_GRP[1].$MCH_POS_Y;
1976: L P[1976] 800cm/min CNT100 COORD PTH ;
:SR[23]=$SCR_GRP[1].$MCH_POS_X;
:SR[24]=$SCR_GRP[1].$MCH_POS_Y;
1977: L P[1977] 800cm/min CNT100 COORD PTH ;
:SR[23]=$SCR_GRP[1].$MCH_POS_X;
:SR[24]=$SCR_GRP[1].$MCH_POS_Y;
1978: L P[1978] 800cm/min CNT100 COORD PTH ;
:SR[23]=$SCR_GRP[1].$MCH_POS_X;
:SR[24]=$SCR_GRP[1].$MCH_POS_Y;
1979: L P[1979] 800cm/min CNT100 COORD PTH ;
:SR[23]=$SCR_GRP[1].$MCH_POS_X;
:SR[24]=$SCR_GRP[1].$MCH_POS_Y;
1980: L P[1980] 800cm/min CNT100 COORD PTH ;
:SR[23]=$SCR_GRP[1].$MCH_POS_X;
:SR[24]=$SCR_GRP[1].$MCH_POS_Y;
1981: L P[1981] 800cm/min CNT100 COORD PTH ;
:SR[23]=$SCR_GRP[1].$MCH_POS_X;
:SR[24]=$SCR_GRP[1].$MCH_POS_Y;
1982: L P[1982] 800cm/min CNT100 COORD PTH ;
:SR[23]=$SCR_GRP[1].$MCH_POS_X;
:SR[24]=$SCR_GRP[1].$MCH_POS_Y;
1983: L P[1983] 800cm/min CNT100 COORD PTH ;
:SR[23]=$SCR_GRP[1].$MCH_POS_X;
:SR[24]=$SCR_GRP[1].$MCH_POS_Y;
1984: L P[1984] 800cm/min CNT100 COORD PTH ;
:SR[23]=$SCR_GRP[1].$MCH_POS_X;
:SR[24]=$SCR_GRP[1].$MCH_POS_Y;
1985: L P[1985] 800cm/min CNT100 COORD PTH ;
:SR[23]=$SCR_GRP[1].$MCH_POS_X;
:SR[24]=$SCR_GRP[1].$MCH_POS_Y;
1986: L P[1986] 800cm/min CNT100 COORD PTH ;
:SR[23]=$SCR_GRP[1].$MCH_POS_X;
:SR[24]=$SCR_GRP[1].$MCH_POS_Y;
